(* CoDeSys 2.3.9.41 project: example.pro *)
(* Libraries: Util.lib 18.5.10 15:14:28, STANDARD.LIB 4.10.05 11:14:46, IECSFC.LIB 13.4.06 15:51:28, SYSLIBTIME.LIB 26.10.21 13:46:42, SYSTASKINFO.LIB 26.10.21 13:46:42, ANALYZATION.LIB 5.10.99 09:05:06, SYSLIBCALLBACK.LIB 26.10.21 13:46:42 *)

(* PLC configuration (modules and I/O channels)
Fast discrete inputs [I_SIMPLE_INPUT] node 0, in %IB0 out %QB0 {ChannellName = Fast discrete inputs; Filtrationtime = 10000}
  AT %IX0.0 [BitInput] Discrete input 1 {ChannellName = Enter name}
  AT %IX0.1 [BitInput] Discrete input 2 {ChannellName = Enter name}
Discrete inputs [ID130] node 1, in %IB1 out %QB1 {ChannellName = Discrete inputs; Filtrationtime_GeneralINP = 16; PinCount = 16}
  discrete_input_first_byte AT %IB1.0 [ByteInput] discrete_input_first_byte {ChannellName = Enter name}
  discrete_input_second_byte AT %IB1.1 [ByteInput] discrete input_second_byte {ChannellName = Enter name}
Fast discrete outputs [OWEN_ID570] node 2, in %IB2 out %QB2 {ChannellName = Fast discrete outputs; SafeValueBool = FALSE; SafeValueBool = FALSE; SafeValueBool = FALSE; SafeValueBool = FALSE}
  hw_run_id1 AT %QX2.0 [BitOutput] Run hot water invertor drive1 {ChannellName = Enter name}
  hw_run_id2 AT %QX2.1 [BitOutput] Run hot water invertor drive2 {ChannellName = Enter name}
  ws_run_id1 AT %QX2.2 [BitOutput] Run water supply invertor drive1 {ChannellName = Enter name}
  ws_run_id2 AT %QX2.3 [BitOutput] Run water supply invertor drive2 {ChannellName = Enter name}
Discrete outputs [ID131] node 3, in %IB3 out %QB3 {ChannellName = Discrete outputs; SafeValueByte = 0; SafeValueByte = 0; SafeValueByteM = 0; PinCount = 24}
  AT %QB3.0 [ByteOutput] 8 discrete outputs {ChannellName = Enter name}
  AT %QB3.1 [ByteOutput] 8 discrete outputs {ChannellName = Enter name}
Special input [ID103] node 4, in %IB4 out %QB4 {ChannellName = Special input}
  AT %IX4.0 [BitInput] Special input {ChannellName = Enter name}
Special output [ID104] node 5, in %IB5 out %QB5 {ChannellName = Special output}
  AT %QX5.0 [BitOutput] Special output {ChannellName = Enter name}
AT %QD6.0 [DWordOutput] Last address {ChannellName = Enter name}
AT %QW6.1 [WordOutput] Last error {ChannellName = Enter name}
RS-485-1 [COM1_USART] node 0, in %IB6.0 out %QB6.0 {ChannellName = RS-485-1; CommunicationSpeed = 115200; Parity = NO PARITY CHECK; BitLength = 8 bits; StopLength = One stop bit; InterfaceType = RS485; FrameOriented = RTU; Timeout = 0; Visibility = No}
AT %QB6.1.0 [ComChannel] Command (0xff - Start) {ChannellName = Enter name}
hw_input_pressure AT %QD6.1.0.0 [FloatOutput] {ChannellName = Enter name}
hw_error_input_pressure AT %QW6.1.1.0 [WordOutput] {ChannellName = Enter name}
hw_output_pressure AT %QD6.1.2.0 [FloatOutput] {ChannellName = Enter name}
hw_error_output_pressure AT %QW6.1.3.0 [WordOutput] {ChannellName = Enter name}
ws_input_pressure AT %QD6.1.4.0 [FloatOutput] {ChannellName = Enter name}
ws_error_input_pressure AT %QW6.1.5.0 [WordOutput] {ChannellName = Enter name}
ws_output_pressure AT %QD6.1.6.0 [FloatOutput] {ChannellName = Enter name}
ws_error_output_pressure AT %QW6.1.7.0 [WordOutput] {ChannellName = Enter name}
ModBus (Master) [MODBUS_MASTER_ID450] node 7, in %IB7 out %QB7 {ChannellName = ModBus (Master); Visibility = No}
  AT %QD7.0 [DWordOutput] Last address {ChannellName = Enter name}
  AT %QW7.1 [WordOutput] Last error {ChannellName = Enter name}
  RS-485-1 [COM1_USART] node 0, in %IB7.0 out %QB7.0 {ChannellName = RS-485-1; CommunicationSpeed = 115200; Parity = NO PARITY CHECK; BitLength = 8 bits; StopLength = One stop bit; InterfaceType = RS485; FrameOriented = RTU; Timeout = 0; Visibility = No}
  Universal Modbus device [ID2000] node 1, in %IB7.1 out %QB7.1 {ChannellName = Universal Modbus device; ModuleIP = 10:0:0:223; ServiceTimeout = 150; TCPport = 502; NetMode = Serial; ModuleSlaveAddress = 32; RequestType = By poll time; PeriodOfService = 100; Visibility = No; RepeatCounter = 0; ByteSequence = Trace_mode}
    AT %QB7.1.0 [ComChannel] Command (0xff - Start) {ChannellName = Enter name}
hw_output_value_id1 AT %QW7.1.0.0 [WordOutput] {ChannellName = Enter name}
hw_output_value_id2 AT %QW7.1.1.0 [WordOutput] {ChannellName = Enter name}
ws_output_value_id1 AT %QW7.1.2.0 [WordOutput] {ChannellName = Enter name}
ws_output_value_id2 AT %QW7.1.3.0 [WordOutput] {ChannellName = Enter name}
AT %QW7.1.4.0 [WordOutput] {ChannellName = Enter name}
AT %QW7.1.5.0 [WordOutput] {ChannellName = Enter name}
AT %QW7.1.6.0 [WordOutput] {ChannellName = Enter name}
AT %QW7.1.7.0 [WordOutput] {ChannellName = Enter name}
Modbus [MODBUS_ID302] node 0, in %IB8.0 out %QB8.0 {ChannellName = Modbus}
  RS-232 [COM2_USART] node 0, in %IB8.0.0 out %QB8.0.0 {ChannellName = RS-232; CommunicationSpeed = 115200; Parity = NO PARITY CHECK; BitLength = 8 bits; StopLength = One stop bit; InterfaceType = RS232; FrameOriented = RTU; Timeout = 0; Visibility = No}
8 bits [8Bit] node 1, in %IB8.1 out %QB8.1 {ChannellName = 8 bit}
  AT %QB8.1.0 [ByteOutput] {ChannellName = Enter name}
8 bits [8Bit] node 2, in %IB8.2 out %QB8.2 {ChannellName = 8 bit}
  AT %QB8.2.0 [ByteOutput] {ChannellName = Enter name}
  AT %QB8.3.0 [ByteOutput] {ChannellName = Enter name}
  AT %QB8.4.0 [ByteOutput] {ChannellName = Enter name}
2 byte [Register] node 5, in %IB8.5 out %QB8.5 {ChannellName = 2 byte}
  hw_pivot_single AT %QW8.5.0 [WordOutput] {ChannellName = Enter name}
2 byte [Register] node 6, in %IB8.6 out %QB8.6 {ChannellName = 2 byte}
  hw_pivot_cascade AT %QW8.6.0 [WordOutput] {ChannellName = Enter name}
2 byte [Register] node 7, in %IB8.7 out %QB8.7 {ChannellName = 2 byte}
  hw_cycle_set_hours AT %QW8.7.0 [WordOutput] {ChannellName = Enter name}
2 byte [Register] node 8, in %IB8.8 out %QB8.8 {ChannellName = 2 byte}
  hw_cycle_set_minutes AT %QW8.8.0 [WordOutput] {ChannellName = Enter name}
2 byte [Register] node 9, in %IB8.9 out %QB8.9 {ChannellName = 2 byte}
  hw_cycle_set_seconds AT %QW8.9.0 [WordOutput] {ChannellName = Enter name}
2 byte [Register] node 10, in %IB8.10 out %QB8.10 {ChannellName = 2 byte}
  hw_cascade_delay_on_hours AT %QW8.10.0 [WordOutput] {ChannellName = Enter name}
2 byte [Register] node 11, in %IB8.11 out %QB8.11 {ChannellName = 2 byte}
  hw_cascade_delay_on_minutes AT %QW8.11.0 [WordOutput] {ChannellName = Enter name}
2 byte [Register] node 12, in %IB8.12 out %QB8.12 {ChannellName = 2 byte}
  hw_cascade_delay_on_seconds AT %QW8.12.0 [WordOutput] {ChannellName = Enter name}
2 byte [Register] node 13, in %IB8.13 out %QB8.13 {ChannellName = 2 byte}
  hw_cascade_delay_off_hours AT %QW8.13.0 [WordOutput] {ChannellName = Enter name}
2 byte [Register] node 14, in %IB8.14 out %QB8.14 {ChannellName = 2 byte}
  hw_cascade_delay_off_minutes AT %QW8.14.0 [WordOutput] {ChannellName = Enter name}
2 byte [Register] node 15, in %IB8.15 out %QB8.15 {ChannellName = 2 byte}
  hw_cascade_delay_off_seconds AT %QW8.15.0 [WordOutput] {ChannellName = Enter name}
2 byte [Register] node 16, in %IB8.16 out %QB8.16 {ChannellName = 2 byte}
  ws_pivot_single AT %QW8.16.0 [WordOutput] {ChannellName = Enter name}
2 byte [Register] node 17, in %IB8.17 out %QB8.17 {ChannellName = 2 byte}
  ws_pivot_cascade AT %QW8.17.0 [WordOutput] {ChannellName = Enter name}
2 byte [Register] node 18, in %IB8.18 out %QB8.18 {ChannellName = 2 byte}
  ws_cycle_set_hours AT %QW8.18.0 [WordOutput] {ChannellName = Enter name}
2 byte [Register] node 19, in %IB8.19 out %QB8.19 {ChannellName = 2 byte}
  ws_cycle_set_minutes AT %QW8.19.0 [WordOutput] {ChannellName = Enter name}
2 byte [Register] node 20, in %IB8.20 out %QB8.20 {ChannellName = 2 byte}
  ws_cycle_set_seconds AT %QW8.20.0 [WordOutput] {ChannellName = Enter name}
2 byte [Register] node 21, in %IB8.21 out %QB8.21 {ChannellName = 2 byte}
  ws_cascade_delay_on_hours AT %QW8.21.0 [WordOutput] {ChannellName = Enter name}
2 byte [Register] node 22, in %IB8.22 out %QB8.22 {ChannellName = 2 byte}
  ws_cascade_delay_on_minutes AT %QW8.22.0 [WordOutput] {ChannellName = Enter name}
2 byte [Register] node 23, in %IB8.23 out %QB8.23 {ChannellName = 2 byte}
  ws_cascade_delay_on_seconds AT %QW8.23.0 [WordOutput] {ChannellName = Enter name}
2 byte [Register] node 24, in %IB8.24 out %QB8.24 {ChannellName = 2 byte}
  ws_cascade_delay_off_hours AT %QW8.24.0 [WordOutput] {ChannellName = Enter name}
2 byte [Register] node 25, in %IB8.25 out %QB8.25 {ChannellName = 2 byte}
  ws_cascade_delay_off_minutes AT %QW8.25.0 [WordOutput] {ChannellName = Enter name}
2 byte [Register] node 26, in %IB8.26 out %QB8.26 {ChannellName = 2 byte}
  ws_cascade_delay_off_seconds AT %QW8.26.0 [WordOutput] {ChannellName = Enter name}
Float [Float] node 27, in %IB8.27 out %QB8.27 {ChannellName = float}
  hw_set_point_pressure AT %QD8.27.0 [FloatOutput] {ChannellName = Enter name}
Float [Float] node 28, in %IB8.28 out %QB8.28 {ChannellName = float}
  ws_set_point_pressure AT %QD8.28.0 [FloatOutput] {ChannellName = Enter name}
Float [Float] node 29, in %IB8.29 out %QB8.29 {ChannellName = float}
  hw_min_measure_range_input AT %QD8.29.0 [FloatOutput] {ChannellName = Enter name}
Float [Float] node 30, in %IB8.30 out %QB8.30 {ChannellName = float}
  hw_max_measure_range_input AT %QD8.30.0 [FloatOutput] {ChannellName = Enter name}
Float [Float] node 31, in %IB8.31 out %QB8.31 {ChannellName = float}
  hw_min_measure_range_output AT %QD8.31.0 [FloatOutput] {ChannellName = Enter name}
Float [Float] node 32, in %IB8.32 out %QB8.32 {ChannellName = float}
  hw_max_measure_range_output AT %QD8.32.0 [FloatOutput] {ChannellName = Enter name}
Float [Float] node 33, in %IB8.33 out %QB8.33 {ChannellName = float}
  ws_min_measure_range_input AT %QD8.33.0 [FloatOutput] {ChannellName = Enter name}
Float [Float] node 34, in %IB8.34 out %QB8.34 {ChannellName = float}
  ws_max_measure_range_input AT %QD8.34.0 [FloatOutput] {ChannellName = Enter name}
Float [Float] node 35, in %IB8.35 out %QB8.35 {ChannellName = float}
  ws_min_measure_range_output AT %QD8.35.0 [FloatOutput] {ChannellName = Enter name}
Float [Float] node 36, in %IB8.36 out %QB8.36 {ChannellName = float}
  ws_max_measure_range_output AT %QD8.36.0 [FloatOutput] {ChannellName = Enter name}
Float [Float] node 37, in %IB8.37 out %QB8.37 {ChannellName = float}
  hw_input_pressure_bar AT %QD8.37.0 [FloatOutput] {ChannellName = Enter name}
Float [Float] node 38, in %IB8.38 out %QB8.38 {ChannellName = float}
  hw_output_pressure_bar AT %QD8.38.0 [FloatOutput] {ChannellName = Enter name}
Float [Float] node 39, in %IB8.39 out %QB8.39 {ChannellName = float}
  ws_input_pressure_bar AT %QD8.39.0 [FloatOutput] {ChannellName = Enter name}
Float [Float] node 40, in %IB8.40 out %QB8.40 {ChannellName = float}
  ws_output_pressure_bar AT %QD8.40.0 [FloatOutput] {ChannellName = Enter name}
Float [Float] node 41, in %IB8.41 out %QB8.41 {ChannellName = float}
  hw_frequency_id1 AT %QD8.41.0 [FloatOutput] {ChannellName = Enter name}
Float [Float] node 42, in %IB8.42 out %QB8.42 {ChannellName = float}
  hw_frequency_id2 AT %QD8.42.0 [FloatOutput] {ChannellName = Enter name}
Float [Float] node 43, in %IB8.43 out %QB8.43 {ChannellName = float}
  ws_frequency_id1 AT %QD8.43.0 [FloatOutput] {ChannellName = Enter name}
Float [Float] node 44, in %IB8.44 out %QB8.44 {ChannellName = float}
  ws_frequency_id2 AT %QD8.44.0 [FloatOutput] {ChannellName = Enter name}
2 byte [Register] node 45, in %IB8.45 out %QB8.45 {ChannellName = 2 byte}
  hw_alarm_error_code AT %QW8.45.0 [WordOutput] {ChannellName = Enter name}
2 byte [Register] node 46, in %IB8.46 out %QB8.46 {ChannellName = 2 byte}
  ws_alarm_error_code AT %QW8.46.0 [WordOutput] {ChannellName = Enter name}
Float [Float] node 47, in %IB8.47 out %QB8.47 {ChannellName = float}
  hw_manual_set_frequency_id1 AT %QD8.47.0 [FloatOutput] {ChannellName = Enter name}
Float [Float] node 48, in %IB8.48 out %QB8.48 {ChannellName = float}
  hw_manual_set_frequency_id2 AT %QD8.48.0 [FloatOutput] {ChannellName = Enter name}
Float [Float] node 49, in %IB8.49 out %QB8.49 {ChannellName = float}
  ws_manual_set_frequency_id1 AT %QD8.49.0 [FloatOutput] {ChannellName = Enter name}
Float [Float] node 50, in %IB8.50 out %QB8.50 {ChannellName = float}
  ws_manual_set_frequency_id2 AT %QD8.50.0 [FloatOutput] {ChannellName = Enter name}
2 byte [Register] node 51, in %IB8.51 out %QB8.51 {ChannellName = 2 byte}
  AT %QW8.51.0 [WordOutput] {ChannellName = Enter name}
2 byte [Register] node 52, in %IB8.52 out %QB8.52 {ChannellName = 2 byte}
  AT %QW8.52.0 [WordOutput] {ChannellName = Enter name}
2 byte [Register] node 53, in %IB8.53 out %QB8.53 {ChannellName = 2 byte}
  AT %QW8.53.0 [WordOutput] {ChannellName = Enter name}
2 byte [Register] node 54, in %IB8.54 out %QB8.54 {ChannellName = 2 byte}
  AT %QW8.54.0 [WordOutput] {ChannellName = Enter name}
2 byte [Register] node 55, in %IB8.55 out %QB8.55 {ChannellName = 2 byte}
  AT %QW8.55.0 [WordOutput] {ChannellName = Enter name}
2 byte [Register] node 56, in %IB8.56 out %QB8.56 {ChannellName = 2 byte}
  AT %QW8.56.0 [WordOutput] {ChannellName = Enter name}
2 byte [Register] node 57, in %IB8.57 out %QB8.57 {ChannellName = 2 byte}
  AT %QW8.57.0 [WordOutput] {ChannellName = Enter name}
2 byte [Register] node 58, in %IB8.58 out %QB8.58 {ChannellName = 2 byte}
  AT %QW8.58.0 [WordOutput] {ChannellName = Enter name}
2 byte [Register] node 59, in %IB8.59 out %QB8.59 {ChannellName = 2 byte}
  AT %QW8.59.0 [WordOutput] {ChannellName = Enter name}
2 byte [Register] node 60, in %IB8.60 out %QB8.60 {ChannellName = 2 byte}
  AT %QW8.60.0 [WordOutput] {ChannellName = Enter name}
2 byte [Register] node 61, in %IB8.61 out %QB8.61 {ChannellName = 2 byte}
  AT %QW8.61.0 [WordOutput] {ChannellName = Enter name}
2 byte [Register] node 62, in %IB8.62 out %QB8.62 {ChannellName = 2 byte}
  AT %QW8.62.0 [WordOutput] {ChannellName = Enter name}
2 byte [Register] node 63, in %IB8.63 out %QB8.63 {ChannellName = 2 byte}
  AT %QW8.63.0 [WordOutput] {ChannellName = Enter name}
2 byte [Register] node 64, in %IB8.64 out %QB8.64 {ChannellName = 2 byte}
  AT %QW8.64.0 [WordOutput] {ChannellName = Enter name}
2 byte [Register] node 65, in %IB8.65 out %QB8.65 {ChannellName = 2 byte}
  AT %QW8.65.0 [WordOutput] {ChannellName = Enter name}
2 byte [Register] node 66, in %IB8.66 out %QB8.66 {ChannellName = 2 byte}
  AT %QW8.66.0 [WordOutput] {ChannellName = Enter name}
2 byte [Register] node 67, in %IB8.67 out %QB8.67 {ChannellName = 2 byte}
  AT %QW8.67.0 [WordOutput] {ChannellName = Enter name}
2 byte [Register] node 68, in %IB8.68 out %QB8.68 {ChannellName = 2 byte}
  AT %QW8.68.0 [WordOutput] {ChannellName = Enter name}
2 byte [Register] node 69, in %IB8.69 out %QB8.69 {ChannellName = 2 byte}
  AT %QW8.69.0 [WordOutput] {ChannellName = Enter name}
2 byte [Register] node 70, in %IB8.70 out %QB8.70 {ChannellName = 2 byte}
  AT %QW8.70.0 [WordOutput] {ChannellName = Enter name}
2 byte [Register] node 71, in %IB8.71 out %QB8.71 {ChannellName = 2 byte}
  AT %QW8.71.0 [WordOutput] {ChannellName = Enter name}
2 byte [Register] node 72, in %IB8.72 out %QB8.72 {ChannellName = 2 byte}
  AT %QW8.72.0 [WordOutput] {ChannellName = Enter name}
2 byte [Register] node 73, in %IB8.73 out %QB8.73 {ChannellName = 2 byte}
  AT %QW8.73.0 [WordOutput] {ChannellName = Enter name}
2 byte [Register] node 74, in %IB8.74 out %QB8.74 {ChannellName = 2 byte}
  AT %QW8.74.0 [WordOutput] {ChannellName = Enter name}
2 byte [Register] node 75, in %IB8.75 out %QB8.75 {ChannellName = 2 byte}
  AT %QW8.75.0 [WordOutput] {ChannellName = Enter name}
2 byte [Register] node 76, in %IB8.76 out %QB8.76 {ChannellName = 2 byte}
  AT %QW8.76.0 [WordOutput] {ChannellName = Enter name}
2 byte [Register] node 77, in %IB8.77 out %QB8.77 {ChannellName = 2 byte}
  AT %QW8.77.0 [WordOutput] {ChannellName = Enter name}
2 byte [Register] node 78, in %IB8.78 out %QB8.78 {ChannellName = 2 byte}
  AT %QW8.78.0 [WordOutput] {ChannellName = Enter name}
2 byte [Register] node 79, in %IB8.79 out %QB8.79 {ChannellName = 2 byte}
  AT %QW8.79.0 [WordOutput] {ChannellName = Enter name}
2 byte [Register] node 80, in %IB8.80 out %QB8.80 {ChannellName = 2 byte}
  AT %QW8.80.0 [WordOutput] {ChannellName = Enter name}
2 byte [Register] node 81, in %IB8.81 out %QB8.81 {ChannellName = 2 byte}
  AT %QW8.81.0 [WordOutput] {ChannellName = Enter name}
2 byte [Register] node 82, in %IB8.82 out %QB8.82 {ChannellName = 2 byte}
  AT %QW8.82.0 [WordOutput] {ChannellName = Enter name}
2 byte [Register] node 83, in %IB8.83 out %QB8.83 {ChannellName = 2 byte}
  AT %QW8.83.0 [WordOutput] {ChannellName = Enter name}
2 byte [Register] node 84, in %IB8.84 out %QB8.84 {ChannellName = 2 byte}
  AT %QW8.84.0 [WordOutput] {ChannellName = Enter name}
2 byte [Register] node 85, in %IB8.85 out %QB8.85 {ChannellName = 2 byte}
  AT %QW8.85.0 [WordOutput] {ChannellName = Enter name}
2 byte [Register] node 86, in %IB8.86 out %QB8.86 {ChannellName = 2 byte}
  AT %QW8.86.0 [WordOutput] {ChannellName = Enter name}
2 byte [Register] node 87, in %IB8.87 out %QB8.87 {ChannellName = 2 byte}
  AT %QW8.87.0 [WordOutput] {ChannellName = Enter name}
2 byte [Register] node 88, in %IB8.88 out %QB8.88 {ChannellName = 2 byte}
  AT %QW8.88.0 [WordOutput] {ChannellName = Enter name}
2 byte [Register] node 89, in %IB8.89 out %QB8.89 {ChannellName = 2 byte}
  AT %QW8.89.0 [WordOutput] {ChannellName = Enter name}
2 byte [Register] node 90, in %IB8.90 out %QB8.90 {ChannellName = 2 byte}
  AT %QW8.90.0 [WordOutput] {ChannellName = Enter name}
2 byte [Register] node 91, in %IB8.91 out %QB8.91 {ChannellName = 2 byte}
  AT %QW8.91.0 [WordOutput] {ChannellName = Enter name}
2 byte [Register] node 92, in %IB8.92 out %QB8.92 {ChannellName = 2 byte}
  AT %QW8.92.0 [WordOutput] {ChannellName = Enter name}
2 byte [Register] node 93, in %IB8.93 out %QB8.93 {ChannellName = 2 byte}
  AT %QW8.93.0 [WordOutput] {ChannellName = Enter name}
2 byte [Register] node 94, in %IB8.94 out %QB8.94 {ChannellName = 2 byte}
  AT %QW8.94.0 [WordOutput] {ChannellName = Enter name}
2 byte [Register] node 95, in %IB8.95 out %QB8.95 {ChannellName = 2 byte}
  AT %QW8.95.0 [WordOutput] {ChannellName = Enter name}
2 byte [Register] node 96, in %IB8.96 out %QB8.96 {ChannellName = 2 byte}
  AT %QW8.96.0 [WordOutput] {ChannellName = Enter name}
2 byte [Register] node 97, in %IB8.97 out %QB8.97 {ChannellName = 2 byte}
  AT %QW8.97.0 [WordOutput] {ChannellName = Enter name}
2 byte [Register] node 98, in %IB8.98 out %QB8.98 {ChannellName = 2 byte}
  AT %QW8.98.0 [WordOutput] {ChannellName = Enter name}
2 byte [Register] node 99, in %IB8.99 out %QB8.99 {ChannellName = 2 byte}
  AT %QW8.99.0 [WordOutput] {ChannellName = Enter name}
2 byte [Register] node 100, in %IB8.100 out %QB8.100 {ChannellName = 2 byte}
  AT %QW8.100.0 [WordOutput] {ChannellName = Enter name}
2 byte [Register] node 101, in %IB8.101 out %QB8.101 {ChannellName = 2 byte}
  AT %QW8.101.0 [WordOutput] {ChannellName = Enter name}
2 byte [Register] node 102, in %IB8.102 out %QB8.102 {ChannellName = 2 byte}
  AT %QW8.102.0 [WordOutput] {ChannellName = Enter name}
2 byte [Register] node 103, in %IB8.103 out %QB8.103 {ChannellName = 2 byte}
  AT %QW8.103.0 [WordOutput] {ChannellName = Enter name}
2 byte [Register] node 104, in %IB8.104 out %QB8.104 {ChannellName = 2 byte}
  AT %QW8.104.0 [WordOutput] {ChannellName = Enter name}
2 byte [Register] node 105, in %IB8.105 out %QB8.105 {ChannellName = 2 byte}
  AT %QW8.105.0 [WordOutput] {ChannellName = Enter name}
2 byte [Register] node 106, in %IB8.106 out %QB8.106 {ChannellName = 2 byte}
  AT %QW8.106.0 [WordOutput] {ChannellName = Enter name}
2 byte [Register] node 107, in %IB8.107 out %QB8.107 {ChannellName = 2 byte}
  AT %QW8.107.0 [WordOutput] {ChannellName = Enter name}
2 byte [Register] node 108, in %IB8.108 out %QB8.108 {ChannellName = 2 byte}
  AT %QW8.108.0 [WordOutput] {ChannellName = Enter name}
2 byte [Register] node 109, in %IB8.109 out %QB8.109 {ChannellName = 2 byte}
  AT %QW8.109.0 [WordOutput] {ChannellName = Enter name}
2 byte [Register] node 110, in %IB8.110 out %QB8.110 {ChannellName = 2 byte}
  AT %QW8.110.0 [WordOutput] {ChannellName = Enter name}
2 byte [Register] node 111, in %IB8.111 out %QB8.111 {ChannellName = 2 byte}
  AT %QW8.111.0 [WordOutput] {ChannellName = Enter name}
2 byte [Register] node 112, in %IB8.112 out %QB8.112 {ChannellName = 2 byte}
  AT %QW8.112.0 [WordOutput] {ChannellName = Enter name}
2 byte [Register] node 113, in %IB8.113 out %QB8.113 {ChannellName = 2 byte}
  AT %QW8.113.0 [WordOutput] {ChannellName = Enter name}
2 byte [Register] node 114, in %IB8.114 out %QB8.114 {ChannellName = 2 byte}
  AT %QW8.114.0 [WordOutput] {ChannellName = Enter name}
2 byte [Register] node 115, in %IB8.115 out %QB8.115 {ChannellName = 2 byte}
  AT %QW8.115.0 [WordOutput] {ChannellName = Enter name}
2 byte [Register] node 116, in %IB8.116 out %QB8.116 {ChannellName = 2 byte}
  AT %QW8.116.0 [WordOutput] {ChannellName = Enter name}
2 byte [Register] node 117, in %IB8.117 out %QB8.117 {ChannellName = 2 byte}
  AT %QW8.117.0 [WordOutput] {ChannellName = Enter name}
2 byte [Register] node 118, in %IB8.118 out %QB8.118 {ChannellName = 2 byte}
  AT %QW8.118.0 [WordOutput] {ChannellName = Enter name}
2 byte [Register] node 119, in %IB8.119 out %QB8.119 {ChannellName = 2 byte}
  AT %QW8.119.0 [WordOutput] {ChannellName = Enter name}
2 byte [Register] node 120, in %IB8.120 out %QB8.120 {ChannellName = 2 byte}
  AT %QW8.120.0 [WordOutput] {ChannellName = Enter name}
2 byte [Register] node 121, in %IB8.121 out %QB8.121 {ChannellName = 2 byte}
  AT %QW8.121.0 [WordOutput] {ChannellName = Enter name}
2 byte [Register] node 122, in %IB8.122 out %QB8.122 {ChannellName = 2 byte}
  AT %QW8.122.0 [WordOutput] {ChannellName = Enter name}
2 byte [Register] node 123, in %IB8.123 out %QB8.123 {ChannellName = 2 byte}
  AT %QW8.123.0 [WordOutput] {ChannellName = Enter name}
2 byte [Register] node 124, in %IB8.124 out %QB8.124 {ChannellName = 2 byte}
  AT %QW8.124.0 [WordOutput] {ChannellName = Enter name}
2 byte [Register] node 125, in %IB8.125 out %QB8.125 {ChannellName = 2 byte}
  AT %QW8.125.0 [WordOutput] {ChannellName = Enter name}
2 byte [Register] node 126, in %IB8.126 out %QB8.126 {ChannellName = 2 byte}
  AT %QW8.126.0 [WordOutput] {ChannellName = Enter name}
2 byte [Register] node 127, in %IB8.127 out %QB8.127 {ChannellName = 2 byte}
  AT %QW8.127.0 [WordOutput] {ChannellName = Enter name}
2 byte [Register] node 128, in %IB8.128 out %QB8.128 {ChannellName = 2 byte}
  AT %QW8.128.0 [WordOutput] {ChannellName = Enter name}
2 byte [Register] node 129, in %IB8.129 out %QB8.129 {ChannellName = 2 byte}
  AT %QW8.129.0 [WordOutput] {ChannellName = Enter name}
2 byte [Register] node 130, in %IB8.130 out %QB8.130 {ChannellName = 2 byte}
  AT %QW8.130.0 [WordOutput] {ChannellName = Enter name}
2 byte [Register] node 131, in %IB8.131 out %QB8.131 {ChannellName = 2 byte}
  AT %QW8.131.0 [WordOutput] {ChannellName = Enter name}
*)

(* Data type in InvertorDrive *)
TYPE classAlarmInvertorDrive :

STRUCT
	external_alarm:STRING(79);
	fault_invertor_drive:STRING(79);
END_STRUCT

END_TYPE

(* Data type in MB110_8U *)
TYPE classAnalogOutputChannel :

STRUCT
	current_value: REAL;
END_STRUCT

END_TYPE

(* Data type in MB110_8U *)
TYPE classAnalogOutputModule :

STRUCT
	channel1:classAnalogOutputChannel;
	channel2:classAnalogOutputChannel;
	channel3:classAnalogOutputChannel;
	channel4:classAnalogOutputChannel;
	channel5:classAnalogOutputChannel;
	channel6:classAnalogOutputChannel;
	channel7:classAnalogOutputChannel;
	channel8:classAnalogOutputChannel;
END_STRUCT

END_TYPE

(* Data type in PLC110/DiscreteInputs *)
TYPE classDiscreteInputByte :

STRUCT
	Bit1:BOOL;
	Bit2:BOOL;
	Bit3:BOOL;
	Bit4:BOOL;
	Bit5:BOOL;
	Bit6:BOOL;
	Bit7:BOOL;
	Bit8:BOOL;
END_STRUCT

END_TYPE

(* Data type in PLC110/DiscreteInputs *)
TYPE classDiscreteInputs :

STRUCT
	first_byte:classDiscreteInputByte;
	second_byte:classDiscreteInputByte;
END_STRUCT

END_TYPE

(* Data type in PLC110/DiscreteOutputs *)
TYPE classDiscreteOutputByte :

STRUCT
	Bit1:BOOL;
	Bit2:BOOL;
	Bit3:BOOL;
	Bit4:BOOL;
	Bit5:BOOL;
	Bit6:BOOL;
	Bit7:BOOL;
	Bit8:BOOL;
END_STRUCT

END_TYPE

(* Data type in PLC110/DiscreteOutputs *)
TYPE classDiscreteOutputs :

STRUCT
	first_byte:classDiscreteOutputByte;
	second_byte:classDiscreteOutputByte;
END_STRUCT

END_TYPE

(* Data type in PLC110/DiscreteInputs *)
TYPE classFastDiscreteInputs :

STRUCT
	Bit1:BOOL;
	Bit2:BOOL;
END_STRUCT

END_TYPE

(* Data type in PLC110/DiscreteOutputs *)
TYPE classFastDiscreteOutputs :

STRUCT
	Bit1:BOOL;
	Bit2:BOOL;
	Bit3:BOOL;
	Bit4:BOOL;
END_STRUCT

END_TYPE

(* Data type in MB110_8A *)
TYPE classInfoAnalogInputChannel :

STRUCT
	current_value:REAL;
	error_message:STRING(79);
END_STRUCT

END_TYPE

(* Data type in MB110_8A *)
TYPE classInfoAnalogInputModule :

STRUCT
	channel1:classInfoAnalogInputChannel;
	channel2:classInfoAnalogInputChannel;
	channel3:classInfoAnalogInputChannel;
	channel4:classInfoAnalogInputChannel;
	channel5:classInfoAnalogInputChannel;
	channel6:classInfoAnalogInputChannel;
	channel7:classInfoAnalogInputChannel;
	channel8:classInfoAnalogInputChannel;
END_STRUCT

END_TYPE

(* Data type in CascadeMode *)
TYPE classInfoCascade :

STRUCT
	pivot:INT;
	error_message:STRING(79);
	error_code: WORD;
	cascade_pump1:classInfoCascadePump;
	cascade_pump2:classInfoCascadePump;
	cascade_pump3:classInfoCascadePump;
	cascade_pump4:classInfoCascadePump;
	cascade_pump5:classInfoCascadePump;
	cascade_pump6:classInfoCascadePump;
	cascade_pump7:classInfoCascadePump;
	cascade_pump8:classInfoCascadePump;
END_STRUCT

END_TYPE

(* Data type in CascadeMode *)
TYPE classInfoCascadePump :

STRUCT
	cascade_pump:BOOL := FALSE;  (*ï¿½ï¿½ï¿½ï¿½ï¿½ï¿½ ï¿½ï¿½ï¿½ï¿½ï¿½ï¿½ ï¿½ï¿½ï¿½ï¿½ï¿½ï¿½*)
	manual:INT := 40;  (*Hz*)
END_STRUCT

END_TYPE

(* Data type in CycleMode *)
TYPE classInfoCycle :

STRUCT
	run_timer: BOOL; (* status work *)
	working_time: TIME; (* pump working time  *)
	pump_number: INT;  (* number working pump *)
	error_code:  WORD;
END_STRUCT

END_TYPE

(* Data type in InvertorDrive *)
TYPE classInfoInvertorDrive :

STRUCT
	active:BOOL;
	status_run:STRING(79);
	set_pid:classSetPid;
	alarm:classAlarmInvertorDrive;
	frequency:REAL;  (* Hz *)
	aout_frequency:REAL;  (* mA *)
	run:BOOL;
	reset_fault:BOOL;
END_STRUCT

END_TYPE

(* Data type in SingleMode *)
TYPE classInfoSingle :
(* class for information single mode. *)

STRUCT
    pivot_pump : INT;
    start_pump : BOOL;
    message: STRING(79);
    error_code: WORD;
END_STRUCT

END_TYPE

(* Data type in InvertorDrive *)
TYPE classInvertorDrive :

STRUCT
	discrete_inputs:classInvertorDriveDiscreteInputs;
	discrete_outputs:classInvertorDriveDiscreteOutputs;
	analog_input:classInvertorDriveAnalogInputs;
	analog_output:classInvertorDriveAnalogOutputs;
	set:classSetInvertorDrive;
	min_frequency:INT;
	max_frequency:INT;
	set_frequency:REAL;
	real_frequency:REAL;(* ï¿½ï¿½ï¿½ï¿½ï¿½ï¿½ï¿½ï¿½ ï¿½ ï¿½ï¿½ï¿½ï¿½ï¿½ï¿½ï¿½ï¿½ï¿½ï¿½ï¿½ ï¿½ï¿½ï¿½ï¿½ï¿½ï¿½ ï¿½ï¿½ï¿½ï¿½ï¿½ï¿½ï¿½ï¿½ï¿½ï¿½ *)
END_STRUCT

END_TYPE

(* Data type in InvertorDrive *)
TYPE classInvertorDriveAnalogInputs :

STRUCT
	set_frequency:REAL;
END_STRUCT

END_TYPE

(* Data type in InvertorDrive *)
TYPE classInvertorDriveAnalogOutputs :

STRUCT
	out_frequency:REAL;
END_STRUCT

END_TYPE

(* Data type in InvertorDrive *)
TYPE classInvertorDriveDiscreteInputs :

STRUCT
	start:BOOL;
	reset_fault:BOOL;
(* external alarm *)
	low_pressure_in:BOOL;
	high_pressure_out:BOOL;
END_STRUCT

END_TYPE

(* Data type in InvertorDrive *)
TYPE classInvertorDriveDiscreteOutputs :

STRUCT
	status_run:BOOL;
	status_alarm:BOOL;
END_STRUCT

END_TYPE

(* Data type in value_scale *)
TYPE classParamsValueScaling :

STRUCT
	in_min: REAL := 0;
	in_max: REAL := 100;
	out_min: REAL := 0;
	out_max: REAL := 100;

END_STRUCT

END_TYPE

(* Data type in PLC110 *)
TYPE classPLC110_32 :

STRUCT
	fast_discrete_inputs:classFastDiscreteInputs;
	discrete_inputs:classDiscreteInputs;
	special_input:classSpecialInput;
	fast_discrete_outputs:classFastDiscreteOutputs;
	discrete_output:classDiscreteOutputs;
	special_output:classSpecialOutput;
END_STRUCT

END_TYPE

(* Data type in PLC110 *)
TYPE classPLC32m2StatusInputs :

STRUCT
	fast_inputs:classFastDiscreteInputs;
	discrete_inputs:classDiscreteInputs;
	special_input:classSpecialInput;
END_STRUCT

END_TYPE

(* Data type in PLC110 *)
TYPE classPLC32m2StatusOutputs :

STRUCT
	fast_outputs:classFastDiscreteOutputs;
	discrete_outputs:classDiscreteOutputs;
	special_output:classSpecialOutput;
END_STRUCT

END_TYPE

(* Data type in MB110_8A *)
TYPE classSetAnalogInputChannel :

STRUCT
	(* ï¿½ï¿½ï¿½ï¿½ï¿½ï¿½ï¿½ï¿½ï¿½ï¿½ï¿½ï¿½ï¿½ï¿½ï¿½ï¿½ ï¿½ï¿½ï¿½ï¿½ï¿½ï¿½ï¿½ï¿½ï¿½ ï¿½ï¿½ï¿½ï¿½ï¿½ï¿½ ï¿½ï¿½ï¿½ï¿½ï¿½ï¿½. ï¿½ï¿½. ï¿½ï¿½ï¿½ï¿½ï¿½ï¿½ï¿½ï¿½ï¿½ï¿½ ï¿½ï¿½ï¿½ï¿½ï¿½ï¿½ï¿½: ï¿½ï¿½ï¿½ï¿½ï¿½ï¿½ï¿½ï¿½ï¿½ï¿½. ï¿½ï¿½ï¿½ï¿½ï¿½ï¿½ï¿½ ï¿½.2 *)
	(* ï¿½ï¿½ï¿½ï¿½ï¿½ï¿½ï¿½ ï¿½ï¿½ï¿½ ï¿½ ï¿½ï¿½ï¿½ï¿½ï¿½ï¿½ï¿½ï¿½ ï¿½ï¿½ ï¿½ï¿½ï¿½ï¿½ï¿½ï¿½ï¿½ï¿½ï¿½: ï¿½ï¿½ï¿½ ï¿½ï¿½ï¿½ï¿½ï¿½ï¿½ï¿½ 4-20mA  *)
	ain_l: REAL := 0;  (* ï¿½ï¿½ï¿½ï¿½ï¿½ï¿½ï¿½ï¿½ Ain.L *)
	ain_h: REAL := 1000;  (* ï¿½ï¿½ï¿½ï¿½ï¿½ï¿½ï¿½ï¿½ Ain.H *)
	analog_min_value: REAL := 4;  (* ï¿½ï¿½ï¿½ï¿½ï¿½ï¿½ï¿½ï¿½ ï¿½ï¿½ï¿½ï¿½ï¿½ï¿½ ï¿½ï¿½ï¿½ï¿½ï¿½ï¿½ï¿½ ï¿½ï¿½ï¿½ï¿½ï¿½ï¿½ï¿½ ï¿½ï¿½ï¿½ï¿½ï¿½ï¿½ï¿½ï¿½ *)
	analog_max_value: REAL := 20;  (* ï¿½ï¿½ï¿½ï¿½ï¿½ï¿½ï¿½ï¿½ ï¿½ï¿½ï¿½ï¿½ï¿½ï¿½ï¿½ ï¿½ï¿½ï¿½ï¿½ï¿½ï¿½ï¿½ ï¿½ï¿½ï¿½ï¿½ï¿½ï¿½ï¿½ ï¿½ï¿½ï¿½ï¿½ï¿½ï¿½ï¿½ï¿½ *)
END_STRUCT

END_TYPE

(* Data type in MB110_8A *)
TYPE classSetAnalogInputsModule :

STRUCT
	ch1_set:classSetAnalogInputChannel;
	ch2_set:classSetAnalogInputChannel;
	ch3_set:classSetAnalogInputChannel;
	ch4_set:classSetAnalogInputChannel;
	ch5_set:classSetAnalogInputChannel;
	ch6_set:classSetAnalogInputChannel;
	ch7_set:classSetAnalogInputChannel;
	ch8_set:classSetAnalogInputChannel;
END_STRUCT

END_TYPE

(* Data type in InvertorDrive/set_auto_invertor_drive *)
TYPE classSetAutoInvertorDrive :

STRUCT
	auto:BOOL := FALSE;
	direct_logic:BOOL := TRUE;  (* ï¿½ï¿½ï¿½ï¿½ ï¿½ï¿½ï¿½ï¿½ï¿½ï¿½ï¿½/ï¿½ï¿½ï¿½ï¿½ï¿½ï¿½ï¿½ï¿½ï¿½ ï¿½ï¿½ï¿½ï¿½ï¿½ï¿½ï¿½ï¿½ï¿½ï¿½; ï¿½ï¿½ï¿½ ï¿½ï¿½ï¿½ï¿½ï¿½ï¿½ï¿½ï¿½ ï¿½ï¿½ï¿½ï¿½ï¿½ï¿½ï¿½ï¿½ï¿½ï¿½ ï¿½ï¿½ï¿½ï¿½ ï¿½ï¿½ï¿½ï¿½ï¿½ï¿½ï¿½ï¿½ ï¿½ï¿½ï¿½ï¿½ï¿½ï¿½ï¿½ï¿½ï¿½ï¿½ï¿½ï¿½ï¿½ï¿½ ï¿½ï¿½ï¿½ï¿½ï¿½ï¿½ï¿½ï¿½ ï¿½ï¿½ï¿½ï¿½ ï¿½ï¿½ï¿½ï¿½ï¿½ï¿½ï¿½, ï¿½ï¿½ï¿½ï¿½ï¿½ï¿½ï¿½ï¿½ ï¿½ï¿½ï¿½ï¿½ï¿½ï¿½ï¿½ ï¿½ï¿½ï¿½ï¿½ï¿½ï¿½ï¿½ï¿½ï¿½ï¿½ï¿½, ï¿½ ï¿½ï¿½ï¿½ï¿½ï¿½ï¿½ï¿½ï¿½*)
	set_point:REAL := 0;  (* ï¿½ï¿½ï¿½ï¿½ï¿½ï¿½ï¿½, ï¿½ï¿½ï¿½ï¿½ï¿½ï¿½ï¿½ï¿½ ï¿½ ï¿½ï¿½ï¿½ï¿½ï¿½ï¿½ï¿½ï¿½ ï¿½ï¿½ï¿½ï¿½ï¿½ï¿½ï¿½ï¿½ï¿½ ï¿½ï¿½ï¿½ï¿½ï¿½ï¿½ï¿½ï¿½ï¿½ï¿½ï¿½ï¿½ï¿½ï¿½ ï¿½ï¿½ï¿½ï¿½ï¿½ï¿½ï¿½ï¿½ *)
	value:REAL := 0;  (* ï¿½ï¿½ï¿½ï¿½ï¿½ï¿½ï¿½ ï¿½ï¿½ï¿½ï¿½ï¿½ï¿½ï¿½ï¿½ ï¿½ï¿½ï¿½ï¿½ï¿½ï¿½ï¿½ï¿½ï¿½ï¿½ï¿½ï¿½ï¿½ï¿½ ï¿½ï¿½ï¿½ï¿½ï¿½ï¿½ï¿½ï¿½, ï¿½ï¿½ï¿½ï¿½ï¿½ï¿½ï¿½ï¿½ï¿½ï¿½ ï¿½ ï¿½ï¿½ï¿½ï¿½ï¿½ï¿½ï¿½ *)
	P:REAL := 2;  (* ï¿½ï¿½ï¿½ï¿½ï¿½ï¿½ï¿½ï¿½ï¿½ï¿½ï¿½ï¿½ï¿½ï¿½ï¿½ï¿½ ï¿½ï¿½ï¿½ï¿½ï¿½ï¿½ï¿½ï¿½ï¿½ï¿½ï¿½ ï¿½ï¿½ï¿½ï¿½ï¿½ï¿½ï¿½ï¿½ï¿½ï¿½, ï¿½ï¿½ï¿½ ï¿½ï¿½ï¿½ï¿½ï¿½ï¿½ï¿½ï¿½ï¿½ï¿½ ï¿½ï¿½ï¿½ï¿½ï¿½ ï¿½ï¿½ï¿½ï¿½ï¿½ï¿½ï¿½ï¿½ï¿½ï¿½ ï¿½ï¿½ï¿½ï¿½ï¿½ï¿½ï¿½ï¿½ï¿½ï¿½ ï¿½ï¿½ï¿½ï¿½ï¿½ï¿½ï¿½*)
	I:INT := 10;  (* ï¿½ï¿½ï¿½ï¿½ï¿½ï¿½ï¿½ï¿½ï¿½ï¿½ï¿½ï¿½ ï¿½ï¿½ï¿½ï¿½ï¿½ï¿½ï¿½ï¿½ï¿½ï¿½ï¿½ ï¿½ï¿½ï¿½ï¿½ï¿½ï¿½ï¿½ï¿½ï¿½ï¿½, ï¿½ï¿½ï¿½ï¿½ï¿½ ï¿½ ï¿½ï¿½ï¿½ï¿½ï¿½ï¿½ï¿½ï¿½ *)
	D:INT := 0;  (* ï¿½ï¿½ï¿½ï¿½ï¿½ï¿½ï¿½ï¿½ï¿½ï¿½ï¿½ï¿½ï¿½ï¿½ï¿½ï¿½ ï¿½ï¿½ï¿½ï¿½ï¿½ï¿½ï¿½ï¿½ï¿½ï¿½ï¿½ ï¿½ï¿½ï¿½ï¿½ï¿½ï¿½ï¿½ï¿½ï¿½ï¿½, ï¿½ï¿½ï¿½ï¿½ï¿½ ï¿½ ï¿½ï¿½ï¿½ï¿½ï¿½ï¿½ï¿½ï¿½ *)
END_STRUCT

END_TYPE

(* Data type in InvertorDrive *)
TYPE classSetInvertorDrive :

STRUCT
	set_auto:classSetAutoInvertorDrive;
	set_frequency:classSetLimitFrequency;
END_STRUCT

END_TYPE

(* Data type in InvertorDrive/set_limit_frequency *)
TYPE classSetLimitFrequency :

STRUCT
	manual:REAL;  (* Hz *)
	min_range:REAL;  (* Hz *)
	max_range:REAL;  (* Hz *)
END_STRUCT

END_TYPE

(* Data type in PID_regulator *)
TYPE classSetPid :

STRUCT
	actual:REAL;
	set_point:REAL;
	P:REAL;  (* ï¿½ï¿½ï¿½ï¿½ï¿½ï¿½ï¿½ï¿½ï¿½ï¿½ï¿½ï¿½ï¿½ï¿½ï¿½ï¿½ ï¿½ï¿½ï¿½ï¿½ï¿½ï¿½ï¿½ï¿½ï¿½ï¿½ï¿½ ï¿½ï¿½ï¿½ï¿½ï¿½ï¿½ï¿½ï¿½ï¿½ï¿½, ï¿½ï¿½ï¿½ ï¿½ï¿½ï¿½ï¿½ï¿½ï¿½ï¿½ï¿½ï¿½ï¿½ ï¿½ï¿½ï¿½ï¿½ï¿½ ï¿½ï¿½ï¿½ï¿½ï¿½ï¿½ï¿½ï¿½ï¿½ï¿½ ï¿½ï¿½ï¿½ï¿½ï¿½ï¿½ï¿½ï¿½ï¿½ï¿½ ï¿½ï¿½ï¿½ï¿½ï¿½ï¿½ï¿½*)
	I:INT;  (* ï¿½ï¿½ï¿½ï¿½ï¿½ï¿½ï¿½ï¿½ï¿½ï¿½ï¿½ï¿½ ï¿½ï¿½ï¿½ï¿½ï¿½ï¿½ï¿½ï¿½ï¿½ï¿½ï¿½ ï¿½ï¿½ï¿½ï¿½ï¿½ï¿½ï¿½ï¿½ï¿½ï¿½, ï¿½ï¿½ï¿½ï¿½ï¿½ ï¿½ ï¿½ï¿½ï¿½ï¿½ï¿½ï¿½ï¿½ï¿½ *)
	D:INT;  (* ï¿½ï¿½ï¿½ï¿½ï¿½ï¿½ï¿½ï¿½ï¿½ï¿½ï¿½ï¿½ï¿½ï¿½ï¿½ï¿½ ï¿½ï¿½ï¿½ï¿½ï¿½ï¿½ï¿½ï¿½ï¿½ï¿½ï¿½ ï¿½ï¿½ï¿½ï¿½ï¿½ï¿½ï¿½ï¿½ï¿½ï¿½, ï¿½ï¿½ï¿½ï¿½ï¿½ ï¿½ ï¿½ï¿½ï¿½ï¿½ï¿½ï¿½ï¿½ï¿½ *)
	Y_manual:REAL := 0;
	Y_offset:REAL;
	Y_min:REAL;
	Y_max:REAL;
	manual:BOOL;
	reset:BOOL;
END_STRUCT

END_TYPE

(* Data type in PressureSensor_4_20ma *)
TYPE classSetPressureSensor4_20 :

STRUCT
	min_measure_range:REAL:=0;
	max_measure_range:REAL:=16;
	min_current_range:REAL:=4;
	max_current_range:REAL:=20;
END_STRUCT

END_TYPE

(* Data type in PLC110/DiscreteInputs *)
TYPE classSpecialInput :

STRUCT
	Bit1:BOOL;
END_STRUCT

END_TYPE

(* Data type in PLC110/DiscreteOutputs *)
TYPE classSpecialOutput :

STRUCT
	Bit1:BOOL;
END_STRUCT

END_TYPE

(* POU PLC_PRG, CFC *)
PROGRAM PLC_PRG
VAR
	PLC: PLC110_32m2;
	analog_inputs_module: MB110_8a;
	currents_value_pack: get_info_analog_outputs_module;
	analog_outputs_module: MY110_8u;
	settings_channel_analog_inputs_module: SetChannelsAnalogInputsModule;
	hw_input: CurrentSensorPressure_4_20;
	hw_output: CurrentSensorPressure_4_20;
	ws_input: CurrentSensorPressure_4_20;
	ws_output: CurrentSensorPressure_4_20;
	(*hw_settings_pressure_input: SetCurrentSensorPressure_4_20;
	hw_settings_pressure_output: SetCurrentSensorPressure_4_20;
	ws_settings_pressure_input: SetCurrentSensorPressure_4_20;
	ws_settings_pressure_output: SetCurrentSensorPressure_4_20;*)
	hw_invertor_drive_1: InvertorDrive;
	hw_invertor_drive_2: InvertorDrive;
	ws_invertor_drive_1: InvertorDrive;
	ws_invertor_drive_2: InvertorDrive;
	hw_settings_pid_id_1: params_in_set_PID;
	hw_settings_pid_id_2: params_in_set_PID;
	ws_settings_pid_id_1: params_in_set_PID;
	ws_settings_pid_id_2: params_in_set_PID;
	pid1: PID;
	pid2: PID;
	pid3: PID;
	pid4: PID;
	 hw_frequency_id_1: REAL;
	hw_frequency_id_2: REAL;
	ws_frequency_id_1: REAL;
	ws_frequency_id_2: REAL;
	(* hw_input_pressure_bar: REAL;
	hw_output_pressure_bar: REAL;
	ws_input_pressure_bar: REAL;
	ws_output_pressure_bar: REAL; *)
	hw_single_mode: Single;
	hw_cycle_mode: cycle;
	hw_cascade_mode: cascade;
	hw_mode_selector: Cascade_Cycle_Selector;
	hw_start_id_1: BOOL;
	hw_start_id_2: BOOL;
	info_analog_inputs_module: classInfoAnalogInputModule;
	hw_info_id_1: classInfoInvertorDrive;
	hw_info_id_2: classInfoInvertorDrive;
	ws_info_id_1: classInfoInvertorDrive;
	ws_info_id_2: classInfoInvertorDrive;
	hw_kpi_35: Kpi;
	hw_kpi_36: Kpi;
	ws_kpi_35: Kpi;
	ws_kpi_36: Kpi;
	plc_inputs: classPLC32m2StatusInputs;
	plc_outputs: classPLC32m2StatusOutputs;
	ws_single_mode: Single;
	ws_cycle_mode: cycle;
	ws_cascade_mode: cascade;
	ws_mode_selector: Cascade_Cycle_Selector;
	ws_start_id_1: BOOL;
	ws_start_id_2: BOOL;
	PLC_110_32_outputs: get_status_outputs;
	out_set_frequency: classParamsValueScaling;
	hw_mode_error: WORD;
	hw_alarm_manager: ALARM_MANAGER;
	(*hw_alarm_on: BOOL;
	ws_alarm_on: BOOL;*)
	ws_mode_error: WORD;
       hw_alarm_message AT %QW8.51.0: STRING(79);
       ws_alarm_message AT %QW8.91.0: STRING(79);

	hw_external_alarm: external_alarm_invertor_drive;
	ws_external_alarm: external_alarm_invertor_drive;
END_VAR

VAR RETAIN
	hw_settings_pressure_input: SetCurrentSensorPressure_4_20;
	hw_settings_pressure_output: SetCurrentSensorPressure_4_20;
	ws_settings_pressure_input: SetCurrentSensorPressure_4_20;
	ws_settings_pressure_output: SetCurrentSensorPressure_4_20;
END_VAR
VAR (* helpers for the ST form of the networks *)
	_t95 : REAL;
	_t97 : REAL;
	_t99 : REAL;
	_t83 : BOOL;
	_t84 : BOOL;
	_t85 : BOOL;
	_t204 : BOOL;
	_t205 : BOOL;
	_t206 : BOOL;
	_t207 : BOOL;
	_t277 : classParamsValueScaling;
	_t190 : REAL;
	_t191 : REAL;
	_t118 : BOOL;
	_t124 : BOOL;
	_t123 : BOOL;
	_t120 : BOOL;
	_t126 : BOOL;
	_t125 : BOOL;
	_t131 : BOOL;
	_t134 : BOOL;
	_t133 : BOOL;
	_t136 : BOOL;
	_t135 : BOOL;
	_t64 : TIME;
	_t65 : TIME;
	_t132 : BOOL;
	_t114 : TIME;
	_t115 : TIME;
	_t300 : BOOL;
	_t334 : BOOL;
END_VAR
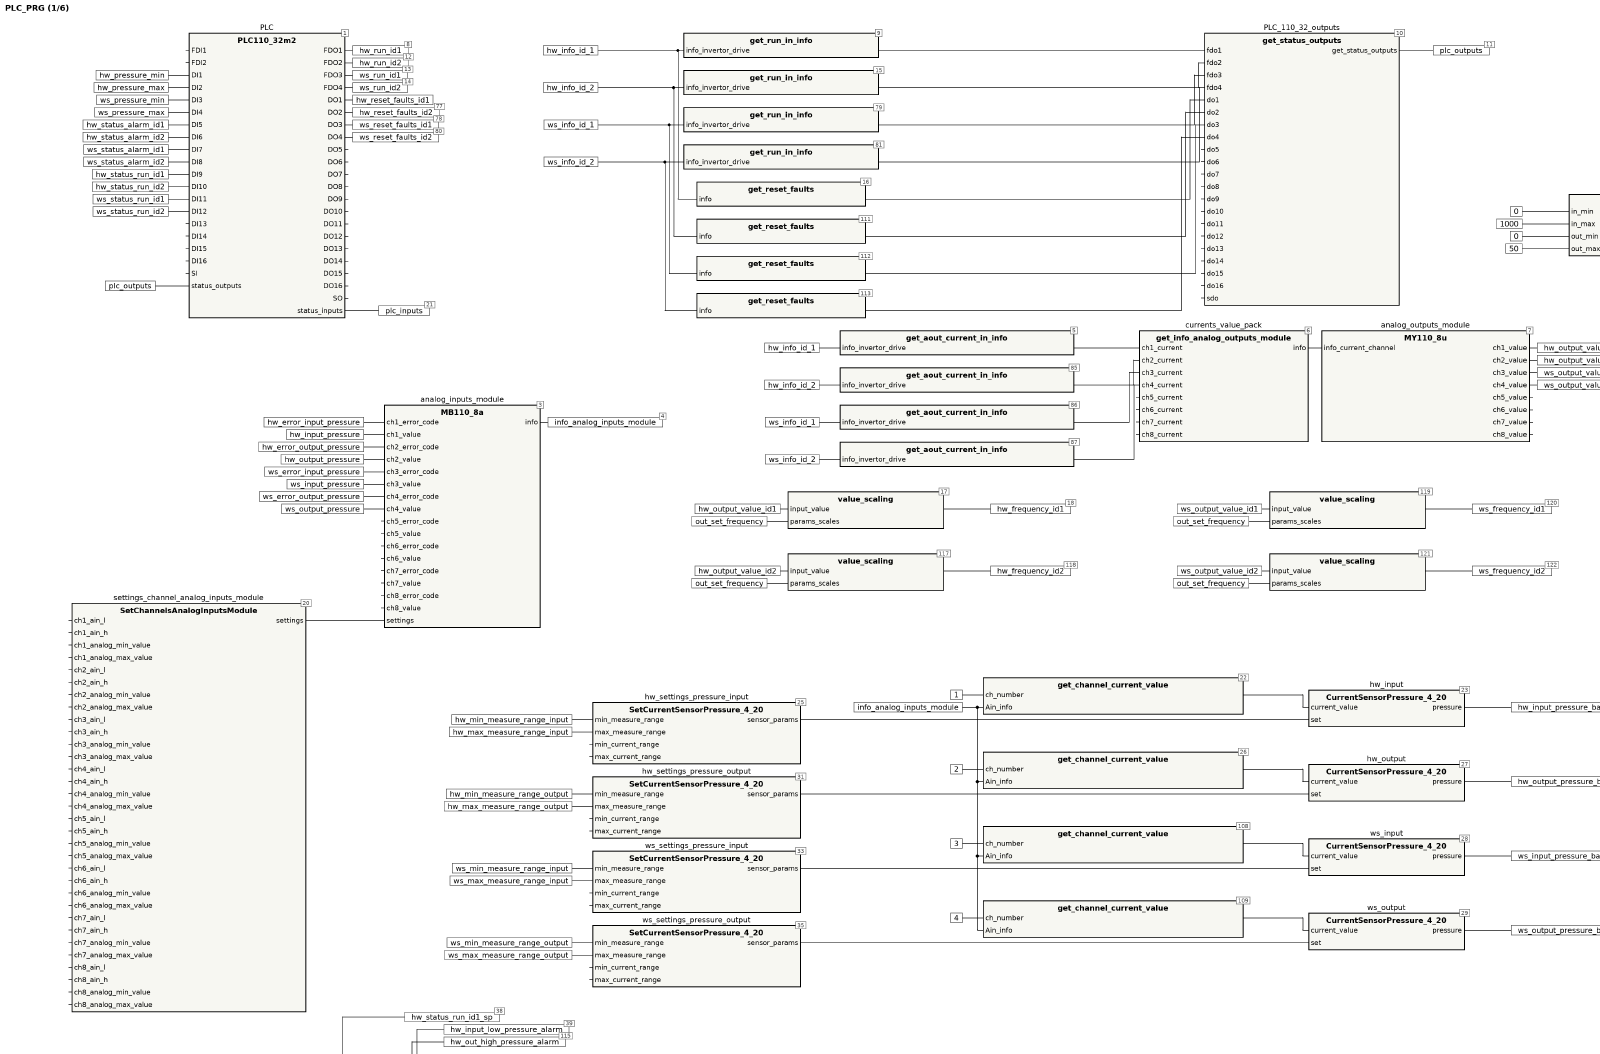
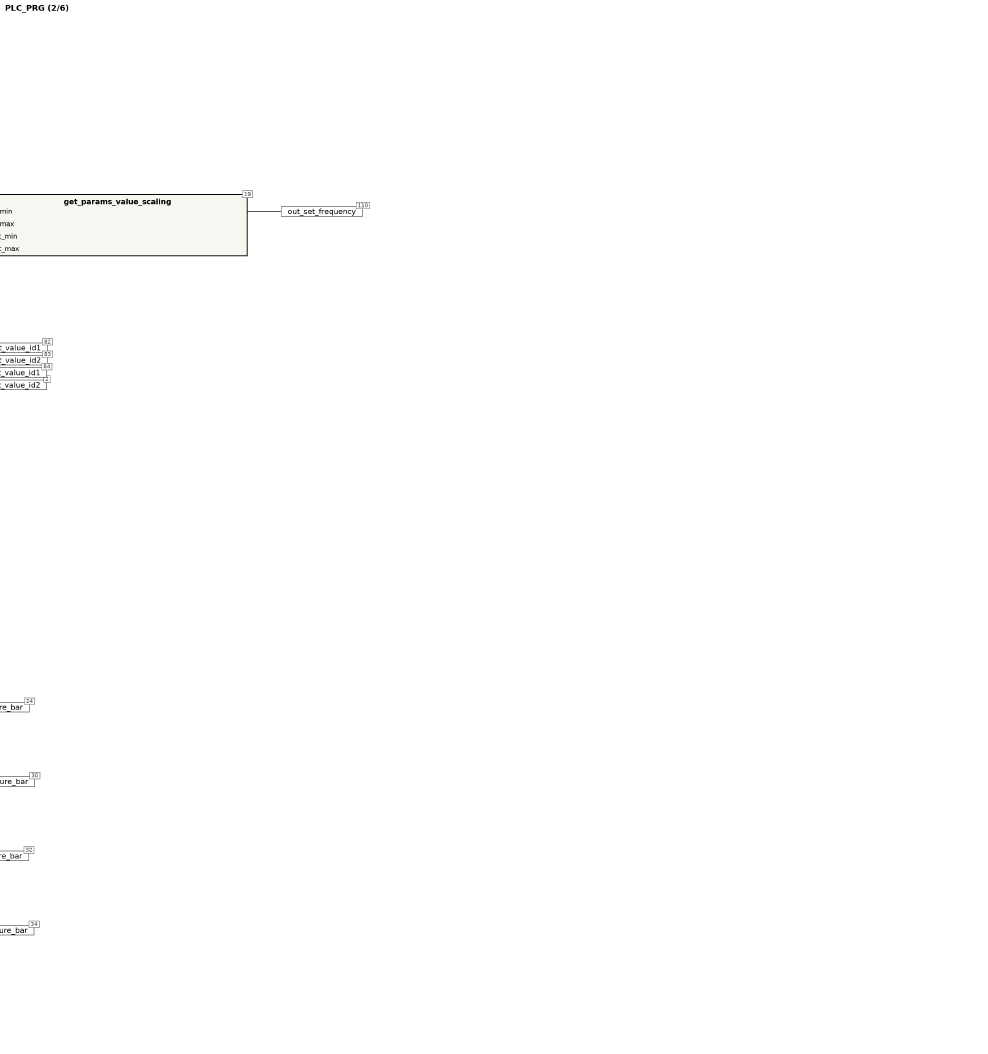
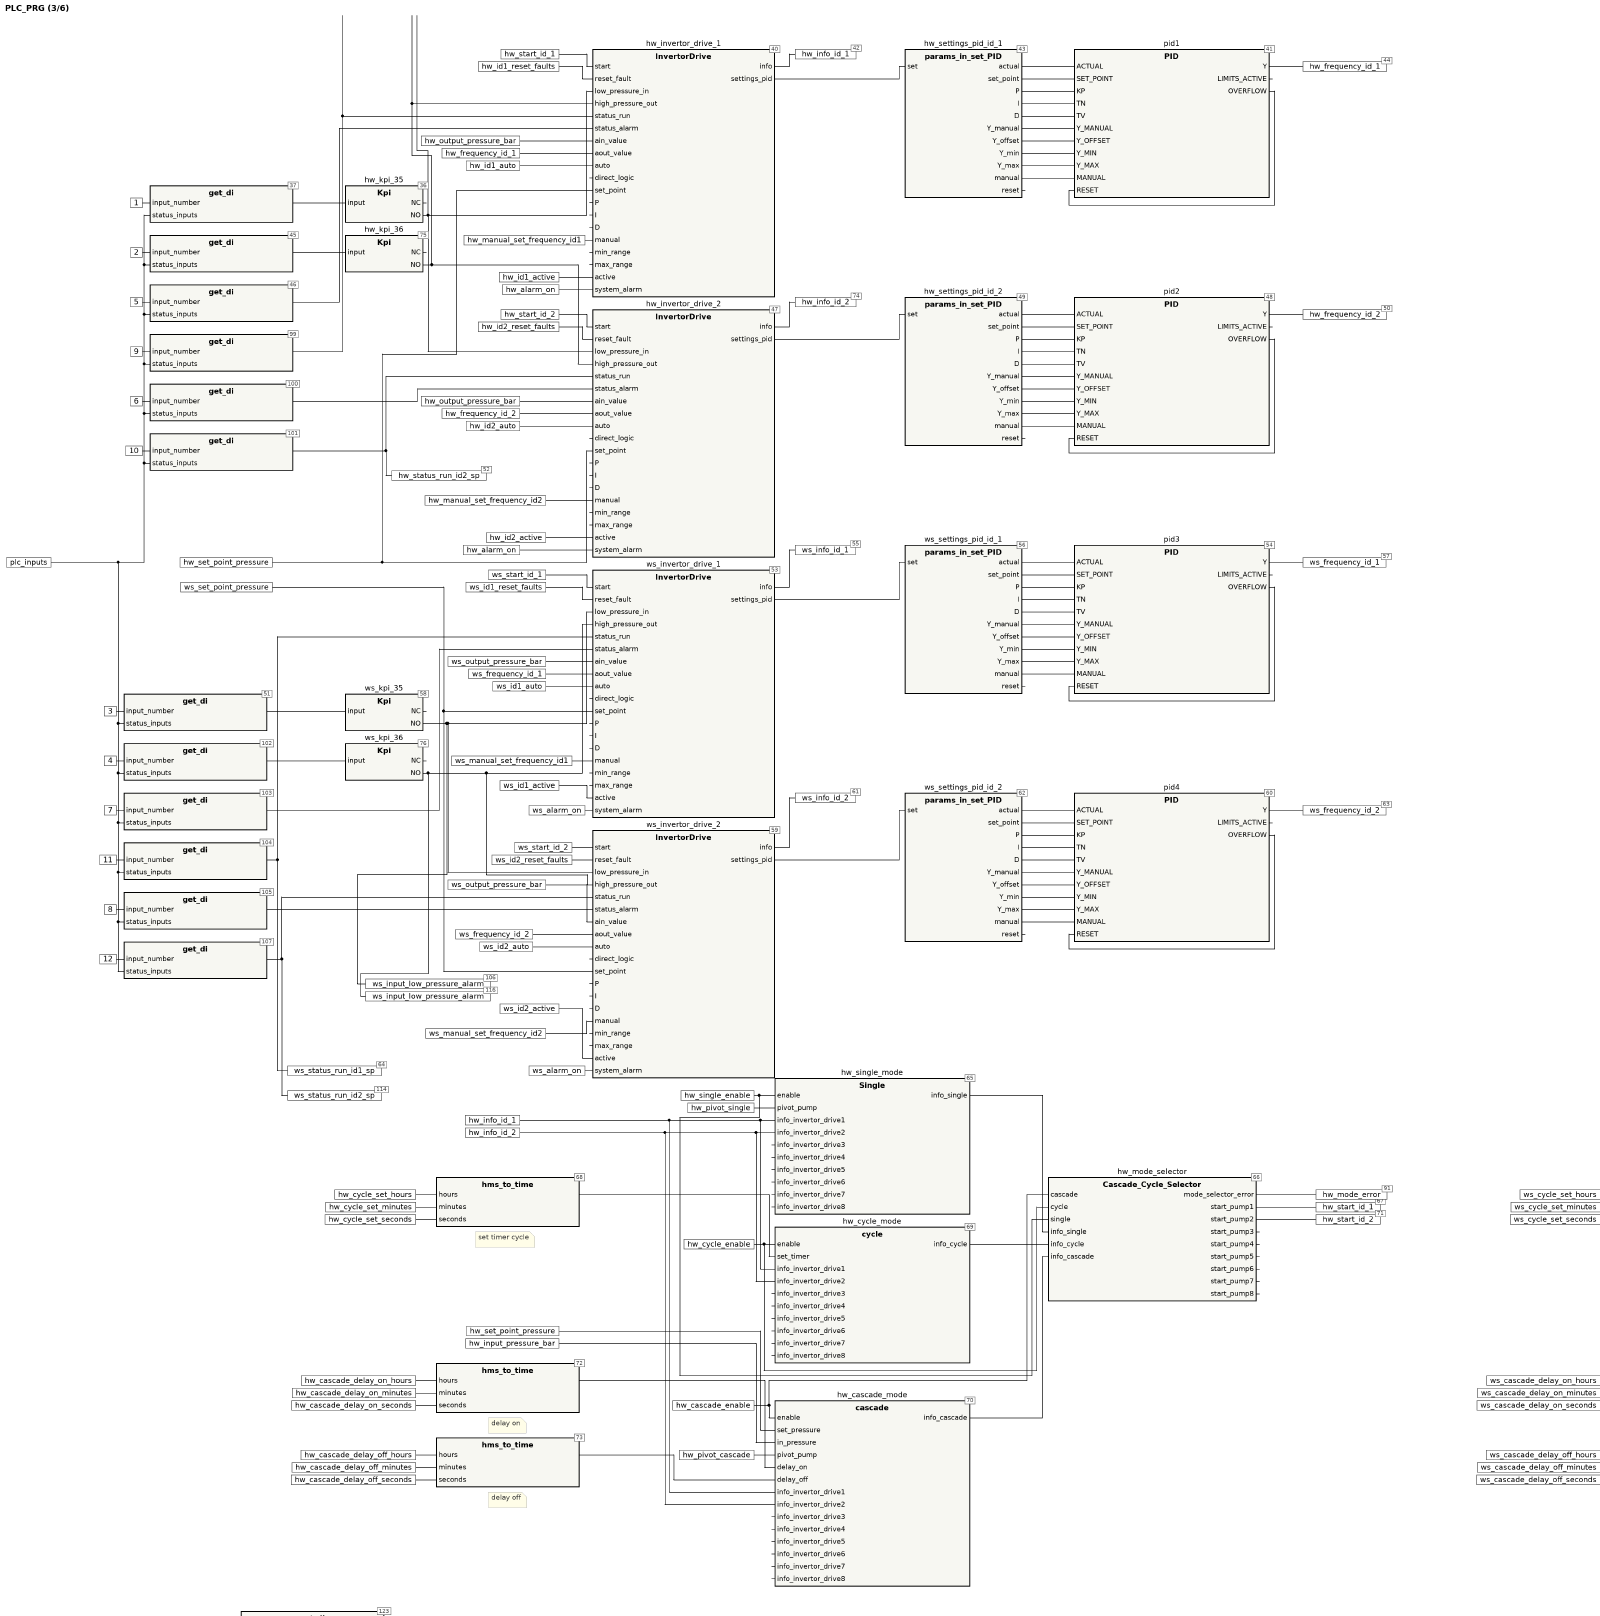
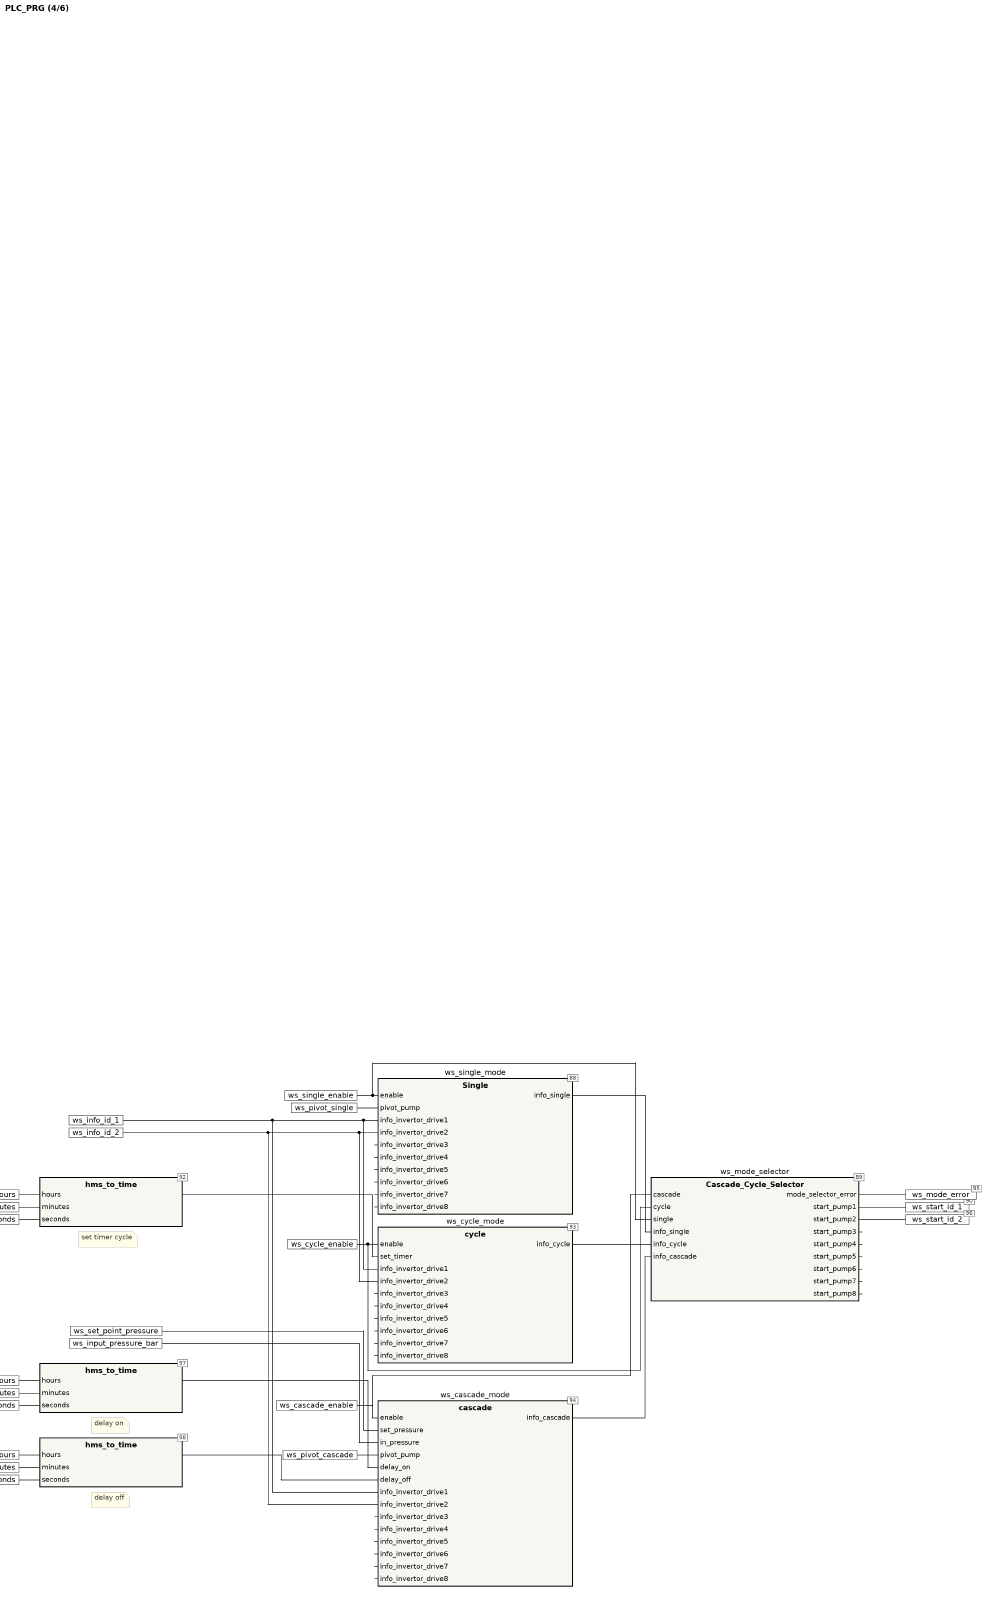
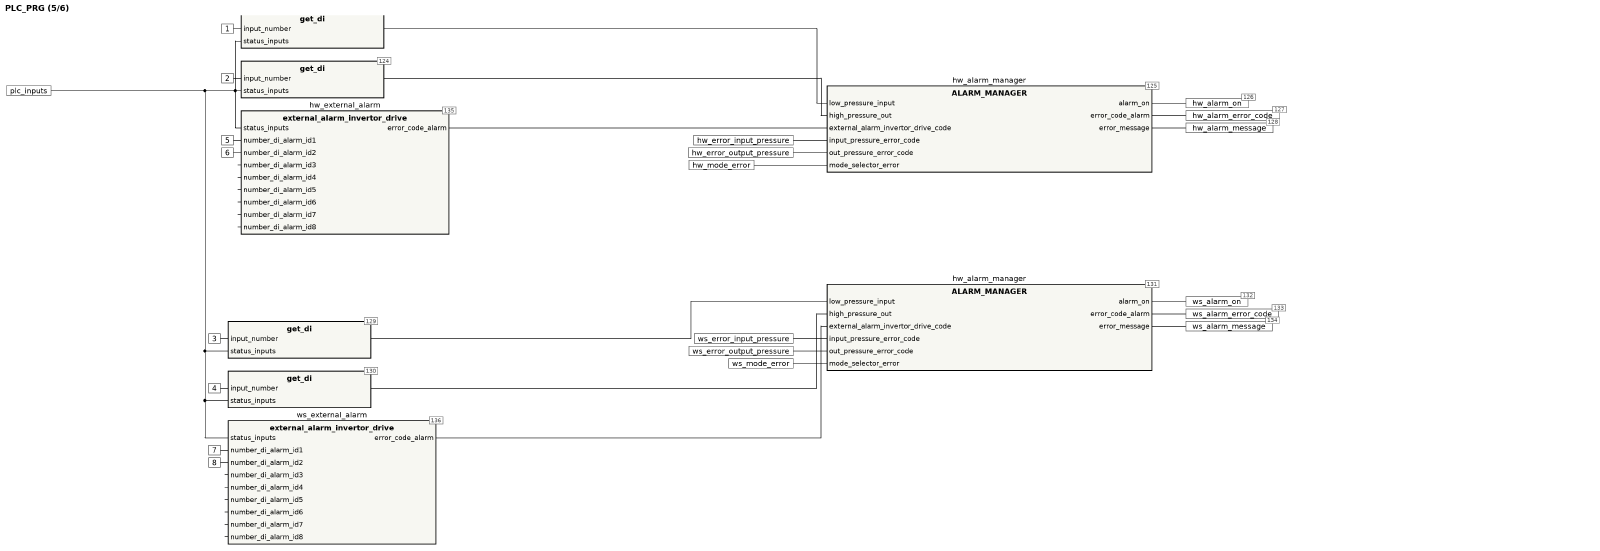
_CFC_ (* Continuous Function Chart, elements in execution order *)
(* set timer cycle *)
(* delay on *)
(* delay off *)
#0 hw_reset_faults_id1 <= #1.DO1
#1 PLC:PLC110_32m2(FDI1: -, FDI2: -, DI1: hw_pressure_min, DI2: hw_pressure_max, DI3: ws_pressure_min, DI4: ws_pressure_max, DI5: hw_status_alarm_id1, DI6: hw_status_alarm_id2, DI7: ws_status_alarm_id1, DI8: ws_status_alarm_id2, DI9: hw_status_run_id1, DI10: hw_status_run_id2, DI11: ws_status_run_id1, DI12: ws_status_run_id2, DI13: -, DI14: -, DI15: -, DI16: -, SI: -, status_outputs: plc_outputs)
#2 ws_output_value_id2 <= #7.ch4_value
#3 analog_inputs_module:MB110_8a(ch1_error_code: hw_error_input_pressure, ch1_value: hw_input_pressure, ch2_error_code: hw_error_output_pressure, ch2_value: hw_output_pressure, ch3_error_code: ws_error_input_pressure, ch3_value: ws_input_pressure, ch4_error_code: ws_error_output_pressure, ch4_value: ws_output_pressure, ch5_error_code: -, ch5_value: -, ch6_error_code: -, ch6_value: -, ch7_error_code: -, ch7_value: -, ch8_error_code: -, ch8_value: -, settings: #20.settings)
#4 info_analog_inputs_module <= #3.info
#5 get_aout_current_in_info(info_invertor_drive: hw_info_id_1)
#6 currents_value_pack:get_info_analog_outputs_module(ch1_current: #5, ch2_current: #85, ch3_current: #86, ch4_current: #87, ch5_current: -, ch6_current: -, ch7_current: -, ch8_current: -)
#7 analog_outputs_module:MY110_8u(info_current_channel: #6.info)
#8 hw_run_id1 <= #1.FDO1
#9 get_run_in_info(info_invertor_drive: hw_info_id_1)
#10 PLC_110_32_outputs:get_status_outputs(fdo1: #9, fdo2: #15, fdo3: #79, fdo4: #81, do1: #16, do2: #111, do3: #112, do4: #113, do5: -, do6: -, do7: -, do8: -, do9: -, do10: -, do11: -, do12: -, do13: -, do14: -, do15: -, do16: -, sdo: -)
#11 plc_outputs <= #10.get_status_outputs
#12 hw_run_id2 <= #1.FDO2
#13 ws_run_id1 <= #1.FDO3
#14 ws_run_id2 <= #1.FDO4
#15 get_run_in_info(info_invertor_drive: hw_info_id_2)
#16 get_reset_faults(info: hw_info_id_1)
#17 value_scaling(input_value: hw_output_value_id1, params_scales: out_set_frequency)
#18 hw_frequency_id1 <= #17
#19 get_params_value_scaling(in_min: 0, in_max: 1000, out_min: 0, out_max: 50)
#20 settings_channel_analog_inputs_module:SetChannelsAnalogInputsModule(ch1_ain_l: -, ch1_ain_h: -, ch1_analog_min_value: -, ch1_analog_max_value: -, ch2_ain_l: -, ch2_ain_h: -, ch2_analog_min_value: -, ch2_analog_max_value: -, ch3_ain_l: -, ch3_ain_h: -, ch3_analog_min_value: -, ch3_analog_max_value: -, ch4_ain_l: -, ch4_ain_h: -, ch4_analog_min_value: -, ch4_analog_max_value: -, ch5_ain_l: -, ch5_ain_h: -, ch5_analog_min_value: -, ch5_analog_max_value: -, ch6_ain_l: -, ch6_ain_h: -, ch6_analog_min_value: -, ch6_analog_max_value: -, ch7_ain_l: -, ch7_ain_h: -, ch7_analog_min_value: -, ch7_analog_max_value: -, ch8_ain_l: -, ch8_ain_h: -, ch8_analog_min_value: -, ch8_analog_max_value: -)
#21 plc_inputs <= #1.status_inputs
#22 get_channel_current_value(ch_number: 1, Ain_info: info_analog_inputs_module)
#23 hw_input:CurrentSensorPressure_4_20(current_value: #22, set: #25.sensor_params)
#24 hw_input_pressure_bar <= #23.pressure
#25 hw_settings_pressure_input:SetCurrentSensorPressure_4_20(min_measure_range: hw_min_measure_range_input, max_measure_range: hw_max_measure_range_input, min_current_range: -, max_current_range: -)
#26 get_channel_current_value(ch_number: 2, Ain_info: info_analog_inputs_module)
#27 hw_output:CurrentSensorPressure_4_20(current_value: #26, set: #31.sensor_params)
#28 ws_input:CurrentSensorPressure_4_20(current_value: #108, set: #33.sensor_params)
#29 ws_output:CurrentSensorPressure_4_20(current_value: #109, set: #35.sensor_params)
#30 hw_output_pressure_bar <= #27.pressure
#31 hw_settings_pressure_output:SetCurrentSensorPressure_4_20(min_measure_range: hw_min_measure_range_output, max_measure_range: hw_max_measure_range_output, min_current_range: -, max_current_range: -)
#32 ws_input_pressure_bar <= #28.pressure
#33 ws_settings_pressure_input:SetCurrentSensorPressure_4_20(min_measure_range: ws_min_measure_range_input, max_measure_range: ws_max_measure_range_input, min_current_range: -, max_current_range: -)
#34 ws_output_pressure_bar <= #29.pressure
#35 ws_settings_pressure_output:SetCurrentSensorPressure_4_20(min_measure_range: ws_min_measure_range_output, max_measure_range: ws_max_measure_range_output, min_current_range: -, max_current_range: -)
#36 hw_kpi_35:Kpi(input: #37)
#37 get_di(input_number: 1, status_inputs: plc_inputs)
#38 hw_status_run_id1_sp <= #99
#39 hw_input_low_pressure_alarm <= #36.NO
#40 hw_invertor_drive_1:InvertorDrive(start: hw_start_id_1, reset_fault: hw_id1_reset_faults, low_pressure_in: #36.NO, high_pressure_out: #75.NO, status_run: #99, status_alarm: #46, ain_value: hw_output_pressure_bar, aout_value: hw_frequency_id_1, auto: hw_id1_auto, direct_logic: -, set_point: hw_set_point_pressure, P: -, I: -, D: -, manual: hw_manual_set_frequency_id1, min_range: -, max_range: -, active: hw_id1_active, system_alarm: hw_alarm_on)
#41 pid1:PID(ACTUAL: #43.actual, SET_POINT: #43.set_point, KP: #43.P, TN: #43.I, TV: #43.D, Y_MANUAL: #43.Y_manual, Y_OFFSET: #43.Y_offset, Y_MIN: #43.Y_min, Y_MAX: #43.Y_max, MANUAL: #43.manual, RESET: #41.OVERFLOW)
#42 hw_info_id_1 <= #40.info
#43 hw_settings_pid_id_1:params_in_set_PID(set: #40.settings_pid)
#44 hw_frequency_id_1 <= #41.Y
#45 get_di(input_number: 2, status_inputs: plc_inputs)
#46 get_di(input_number: 5, status_inputs: plc_inputs)
#47 hw_invertor_drive_2:InvertorDrive(start: hw_start_id_2, reset_fault: hw_id2_reset_faults, low_pressure_in: #36.NO, high_pressure_out: #75.NO, status_run: #101, status_alarm: #100, ain_value: hw_output_pressure_bar, aout_value: hw_frequency_id_2, auto: hw_id2_auto, direct_logic: -, set_point: hw_set_point_pressure, P: -, I: -, D: -, manual: hw_manual_set_frequency_id2, min_range: -, max_range: -, active: hw_id2_active, system_alarm: hw_alarm_on)
#48 pid2:PID(ACTUAL: #49.actual, SET_POINT: #49.set_point, KP: #49.P, TN: #49.I, TV: #49.D, Y_MANUAL: #49.Y_manual, Y_OFFSET: #49.Y_offset, Y_MIN: #49.Y_min, Y_MAX: #49.Y_max, MANUAL: #49.manual, RESET: #48.OVERFLOW)
#49 hw_settings_pid_id_2:params_in_set_PID(set: #47.settings_pid)
#50 hw_frequency_id_2 <= #48.Y
#51 get_di(input_number: 3, status_inputs: plc_inputs)
#52 hw_status_run_id2_sp <= #101
#53 ws_invertor_drive_1:InvertorDrive(start: ws_start_id_1, reset_fault: ws_id1_reset_faults, low_pressure_in: #58.NO, high_pressure_out: #76.NO, status_run: #104, status_alarm: #103, ain_value: ws_output_pressure_bar, aout_value: ws_frequency_id_1, auto: ws_id1_auto, direct_logic: -, set_point: ws_set_point_pressure, P: -, I: -, D: -, manual: ws_manual_set_frequency_id1, min_range: -, max_range: -, active: ws_id1_active, system_alarm: ws_alarm_on)
#54 pid3:PID(ACTUAL: #56.actual, SET_POINT: #56.set_point, KP: #56.P, TN: #56.I, TV: #56.D, Y_MANUAL: #56.Y_manual, Y_OFFSET: #56.Y_offset, Y_MIN: #56.Y_min, Y_MAX: #56.Y_max, MANUAL: #56.manual, RESET: #54.OVERFLOW)
#55 ws_info_id_1 <= #53.info
#56 ws_settings_pid_id_1:params_in_set_PID(set: #53.settings_pid)
#57 ws_frequency_id_1 <= #54.Y
#58 ws_kpi_35:Kpi(input: #51)
#59 ws_invertor_drive_2:InvertorDrive(start: ws_start_id_2, reset_fault: ws_id2_reset_faults, low_pressure_in: #58.NO, high_pressure_out: #76.NO, status_run: #107, status_alarm: #105, ain_value: ws_output_pressure_bar, aout_value: ws_frequency_id_2, auto: ws_id2_auto, direct_logic: -, set_point: ws_set_point_pressure, P: -, I: -, D: -, manual: ws_manual_set_frequency_id2, min_range: -, max_range: -, active: ws_id2_active, system_alarm: ws_alarm_on)
#60 pid4:PID(ACTUAL: #62.actual, SET_POINT: #62.set_point, KP: #62.P, TN: #62.I, TV: #62.D, Y_MANUAL: #62.Y_manual, Y_OFFSET: #62.Y_offset, Y_MIN: #62.Y_min, Y_MAX: #62.Y_max, MANUAL: #62.manual, RESET: #60.OVERFLOW)
#61 ws_info_id_2 <= #59.info
#62 ws_settings_pid_id_2:params_in_set_PID(set: #59.settings_pid)
#63 ws_frequency_id_2 <= #60.Y
#64 ws_status_run_id1_sp <= #104
#65 hw_single_mode:Single(enable: hw_single_enable, pivot_pump: hw_pivot_single, info_invertor_drive1: hw_info_id_1, info_invertor_drive2: hw_info_id_2, info_invertor_drive3: -, info_invertor_drive4: -, info_invertor_drive5: -, info_invertor_drive6: -, info_invertor_drive7: -, info_invertor_drive8: -)
#66 hw_mode_selector:Cascade_Cycle_Selector(cascade: hw_cascade_enable, cycle: hw_cycle_enable, single: hw_single_enable, info_single: #65.info_single, info_cycle: #69.info_cycle, info_cascade: #70.info_cascade)
#67 hw_start_id_1 <= #66.start_pump1
#68 hms_to_time(hours: hw_cycle_set_hours, minutes: hw_cycle_set_minutes, seconds: hw_cycle_set_seconds)
#69 hw_cycle_mode:cycle(enable: hw_cycle_enable, set_timer: #68, info_invertor_drive1: hw_info_id_1, info_invertor_drive2: hw_info_id_2, info_invertor_drive3: -, info_invertor_drive4: -, info_invertor_drive5: -, info_invertor_drive6: -, info_invertor_drive7: -, info_invertor_drive8: -)
#70 hw_cascade_mode:cascade(enable: hw_cascade_enable, set_pressure: hw_set_point_pressure, in_pressure: hw_input_pressure_bar, pivot_pump: hw_pivot_cascade, delay_on: #72, delay_off: #73, info_invertor_drive1: hw_info_id_1, info_invertor_drive2: hw_info_id_2, info_invertor_drive3: -, info_invertor_drive4: -, info_invertor_drive5: -, info_invertor_drive6: -, info_invertor_drive7: -, info_invertor_drive8: -)
#71 hw_start_id_2 <= #66.start_pump2
#72 hms_to_time(hours: hw_cascade_delay_on_hours, minutes: hw_cascade_delay_on_minutes, seconds: hw_cascade_delay_on_seconds)
#73 hms_to_time(hours: hw_cascade_delay_off_hours, minutes: hw_cascade_delay_off_minutes, seconds: hw_cascade_delay_off_seconds)
#74 hw_info_id_2 <= #47.info
#75 hw_kpi_36:Kpi(input: #45)
#76 ws_kpi_36:Kpi(input: #102)
#77 hw_reset_faults_id2 <= #1.DO2
#78 ws_reset_faults_id1 <= #1.DO3
#79 get_run_in_info(info_invertor_drive: ws_info_id_1)
#80 ws_reset_faults_id2 <= #1.DO4
#81 get_run_in_info(info_invertor_drive: ws_info_id_2)
#82 hw_output_value_id1 <= #7.ch1_value
#83 hw_output_value_id2 <= #7.ch2_value
#84 ws_output_value_id1 <= #7.ch3_value
#85 get_aout_current_in_info(info_invertor_drive: hw_info_id_2)
#86 get_aout_current_in_info(info_invertor_drive: ws_info_id_1)
#87 get_aout_current_in_info(info_invertor_drive: ws_info_id_2)
(* set timer cycle *)
(* delay on *)
(* delay off *)
#88 ws_single_mode:Single(enable: ws_single_enable, pivot_pump: ws_pivot_single, info_invertor_drive1: ws_info_id_1, info_invertor_drive2: ws_info_id_2, info_invertor_drive3: -, info_invertor_drive4: -, info_invertor_drive5: -, info_invertor_drive6: -, info_invertor_drive7: -, info_invertor_drive8: -)
#89 ws_mode_selector:Cascade_Cycle_Selector(cascade: ws_cascade_enable, cycle: ws_cycle_enable, single: ws_single_enable, info_single: #88.info_single, info_cycle: #93.info_cycle, info_cascade: #94.info_cascade)
#90 ws_start_id_1 <= #89.start_pump1
#91 hw_mode_error <= #66.mode_selector_error
#92 hms_to_time(hours: ws_cycle_set_hours, minutes: ws_cycle_set_minutes, seconds: ws_cycle_set_seconds)
#93 ws_cycle_mode:cycle(enable: ws_cycle_enable, set_timer: #92, info_invertor_drive1: ws_info_id_1, info_invertor_drive2: ws_info_id_2, info_invertor_drive3: -, info_invertor_drive4: -, info_invertor_drive5: -, info_invertor_drive6: -, info_invertor_drive7: -, info_invertor_drive8: -)
#94 ws_cascade_mode:cascade(enable: ws_cascade_enable, set_pressure: ws_set_point_pressure, in_pressure: ws_input_pressure_bar, pivot_pump: ws_pivot_cascade, delay_on: #97, delay_off: #98, info_invertor_drive1: ws_info_id_1, info_invertor_drive2: ws_info_id_2, info_invertor_drive3: -, info_invertor_drive4: -, info_invertor_drive5: -, info_invertor_drive6: -, info_invertor_drive7: -, info_invertor_drive8: -)
#95 ws_mode_error <= #89.mode_selector_error
#96 ws_start_id_2 <= #89.start_pump2
#97 hms_to_time(hours: ws_cascade_delay_on_hours, minutes: ws_cascade_delay_on_minutes, seconds: ws_cascade_delay_on_seconds)
#98 hms_to_time(hours: ws_cascade_delay_off_hours, minutes: ws_cascade_delay_off_minutes, seconds: ws_cascade_delay_off_seconds)
#99 get_di(input_number: 9, status_inputs: plc_inputs)
#100 get_di(input_number: 6, status_inputs: plc_inputs)
#101 get_di(input_number: 10, status_inputs: plc_inputs)
#102 get_di(input_number: 4, status_inputs: plc_inputs)
#103 get_di(input_number: 7, status_inputs: plc_inputs)
#104 get_di(input_number: 11, status_inputs: plc_inputs)
#105 get_di(input_number: 8, status_inputs: plc_inputs)
#106 ws_input_low_pressure_alarm <= #58.NO
#107 get_di(input_number: 12, status_inputs: plc_inputs)
#108 get_channel_current_value(ch_number: 3, Ain_info: info_analog_inputs_module)
#109 get_channel_current_value(ch_number: 4, Ain_info: info_analog_inputs_module)
#110 out_set_frequency <= #19
#111 get_reset_faults(info: hw_info_id_2)
#112 get_reset_faults(info: ws_info_id_1)
#113 get_reset_faults(info: ws_info_id_2)
#114 ws_status_run_id2_sp <= #107
#115 hw_out_high_pressure_alarm <= #75.NO
#116 ws_input_low_pressure_alarm <= #76.NO
#117 value_scaling(input_value: hw_output_value_id2, params_scales: out_set_frequency)
#118 hw_frequency_id2 <= #117
#119 value_scaling(input_value: ws_output_value_id1, params_scales: out_set_frequency)
#120 ws_frequency_id1 <= #119
#121 value_scaling(input_value: ws_output_value_id2, params_scales: out_set_frequency)
#122 ws_frequency_id2 <= #121
#123 get_di(input_number: 1, status_inputs: plc_inputs)
#124 get_di(input_number: 2, status_inputs: plc_inputs)
#125 hw_alarm_manager:ALARM_MANAGER(low_pressure_input: #123, high_pressure_out: #124, external_alarm_invertor_drive_code: #135.error_code_alarm, input_pressure_error_code: hw_error_input_pressure, out_pressure_error_code: hw_error_output_pressure, mode_selector_error: hw_mode_error)
#126 hw_alarm_on <= #125.alarm_on
#127 hw_alarm_error_code <= #125.error_code_alarm
#128 hw_alarm_message <= #125.error_message
#129 get_di(input_number: 3, status_inputs: plc_inputs)
#130 get_di(input_number: 4, status_inputs: plc_inputs)
#131 hw_alarm_manager:ALARM_MANAGER(low_pressure_input: #129, high_pressure_out: #130, external_alarm_invertor_drive_code: #136.error_code_alarm, input_pressure_error_code: ws_error_input_pressure, out_pressure_error_code: ws_error_output_pressure, mode_selector_error: ws_mode_error)
#132 ws_alarm_on <= #131.alarm_on
#133 ws_alarm_error_code <= #131.error_code_alarm
#134 ws_alarm_message <= #131.error_message
#135 hw_external_alarm:external_alarm_invertor_drive(status_inputs: plc_inputs, number_di_alarm_id1: 5, number_di_alarm_id2: 6, number_di_alarm_id3: -, number_di_alarm_id4: -, number_di_alarm_id5: -, number_di_alarm_id6: -, number_di_alarm_id7: -, number_di_alarm_id8: -)
#136 ws_external_alarm:external_alarm_invertor_drive(status_inputs: plc_inputs, number_di_alarm_id1: 7, number_di_alarm_id2: 8, number_di_alarm_id3: -, number_di_alarm_id4: -, number_di_alarm_id5: -, number_di_alarm_id6: -, number_di_alarm_id7: -, number_di_alarm_id8: -)
_END_CFC_
(* the same logic as Structured Text *)
(* set timer cycle *)
(* delay on *)
(* delay off *)
hw_reset_faults_id1 := PLC.DO1;
PLC(DI1 := hw_pressure_min, DI2 := hw_pressure_max, DI3 := ws_pressure_min, DI4 := ws_pressure_max, DI5 := hw_status_alarm_id1, DI6 := hw_status_alarm_id2, DI7 := ws_status_alarm_id1, DI8 := ws_status_alarm_id2, DI9 := hw_status_run_id1, DI10 := hw_status_run_id2, DI11 := ws_status_run_id1, DI12 := ws_status_run_id2, status_outputs := plc_outputs);
ws_output_value_id2 := analog_outputs_module.ch4_value;
analog_inputs_module(ch1_error_code := hw_error_input_pressure, ch1_value := hw_input_pressure, ch2_error_code := hw_error_output_pressure, ch2_value := hw_output_pressure, ch3_error_code := ws_error_input_pressure, ch3_value := ws_input_pressure, ch4_error_code := ws_error_output_pressure, ch4_value := ws_output_pressure, settings := settings_channel_analog_inputs_module.settings);
info_analog_inputs_module := analog_inputs_module.info;
currents_value_pack(ch1_current := get_aout_current_in_info(info_invertor_drive := hw_info_id_1), ch2_current := _t95, ch3_current := _t97, ch4_current := _t99);
analog_outputs_module(info_current_channel := currents_value_pack.info);
hw_run_id1 := PLC.FDO1;
PLC_110_32_outputs(fdo1 := get_run_in_info(info_invertor_drive := hw_info_id_1), fdo2 := _t83, fdo3 := _t84, fdo4 := _t85, do1 := _t204, do2 := _t205, do3 := _t206, do4 := _t207);
plc_outputs := PLC_110_32_outputs.get_status_outputs;
hw_run_id2 := PLC.FDO2;
ws_run_id1 := PLC.FDO3;
ws_run_id2 := PLC.FDO4;
_t83 := get_run_in_info(info_invertor_drive := hw_info_id_2);
_t204 := get_reset_faults(info := hw_info_id_1);
hw_frequency_id1 := value_scaling(input_value := hw_output_value_id1, params_scales := out_set_frequency);
_t277 := get_params_value_scaling(in_min := 0, in_max := 1000, out_min := 0, out_max := 50);
settings_channel_analog_inputs_module();
plc_inputs := PLC.status_inputs;
hw_input(current_value := get_channel_current_value(ch_number := 1, Ain_info := info_analog_inputs_module), set := hw_settings_pressure_input.sensor_params);
hw_input_pressure_bar := hw_input.pressure;
hw_settings_pressure_input(min_measure_range := hw_min_measure_range_input, max_measure_range := hw_max_measure_range_input);
hw_output(current_value := get_channel_current_value(ch_number := 2, Ain_info := info_analog_inputs_module), set := hw_settings_pressure_output.sensor_params);
ws_input(current_value := _t190, set := ws_settings_pressure_input.sensor_params);
ws_output(current_value := _t191, set := ws_settings_pressure_output.sensor_params);
hw_output_pressure_bar := hw_output.pressure;
hw_settings_pressure_output(min_measure_range := hw_min_measure_range_output, max_measure_range := hw_max_measure_range_output);
ws_input_pressure_bar := ws_input.pressure;
ws_settings_pressure_input(min_measure_range := ws_min_measure_range_input, max_measure_range := ws_max_measure_range_input);
ws_output_pressure_bar := ws_output.pressure;
ws_settings_pressure_output(min_measure_range := ws_min_measure_range_output, max_measure_range := ws_max_measure_range_output);
hw_kpi_35(input := _t118);
_t118 := get_di(input_number := 1, status_inputs := plc_inputs);
hw_status_run_id1_sp := _t124;
hw_input_low_pressure_alarm := hw_kpi_35.NO;
hw_invertor_drive_1(start := hw_start_id_1, reset_fault := hw_id1_reset_faults, low_pressure_in := hw_kpi_35.NO, high_pressure_out := hw_kpi_36.NO, status_run := _t124, status_alarm := _t123, ain_value := hw_output_pressure_bar, aout_value := hw_frequency_id_1, auto := hw_id1_auto, set_point := hw_set_point_pressure, manual := hw_manual_set_frequency_id1, active := hw_id1_active, system_alarm := hw_alarm_on);
pid1(ACTUAL := hw_settings_pid_id_1.actual, SET_POINT := hw_settings_pid_id_1.set_point, KP := hw_settings_pid_id_1.P, TN := hw_settings_pid_id_1.I, TV := hw_settings_pid_id_1.D, Y_MANUAL := hw_settings_pid_id_1.Y_manual, Y_OFFSET := hw_settings_pid_id_1.Y_offset, Y_MIN := hw_settings_pid_id_1.Y_min, Y_MAX := hw_settings_pid_id_1.Y_max, MANUAL := hw_settings_pid_id_1.manual, RESET := pid1.OVERFLOW);
hw_info_id_1 := hw_invertor_drive_1.info;
hw_settings_pid_id_1(set := hw_invertor_drive_1.settings_pid);
hw_frequency_id_1 := pid1.Y;
_t120 := get_di(input_number := 2, status_inputs := plc_inputs);
_t123 := get_di(input_number := 5, status_inputs := plc_inputs);
hw_invertor_drive_2(start := hw_start_id_2, reset_fault := hw_id2_reset_faults, low_pressure_in := hw_kpi_35.NO, high_pressure_out := hw_kpi_36.NO, status_run := _t126, status_alarm := _t125, ain_value := hw_output_pressure_bar, aout_value := hw_frequency_id_2, auto := hw_id2_auto, set_point := hw_set_point_pressure, manual := hw_manual_set_frequency_id2, active := hw_id2_active, system_alarm := hw_alarm_on);
pid2(ACTUAL := hw_settings_pid_id_2.actual, SET_POINT := hw_settings_pid_id_2.set_point, KP := hw_settings_pid_id_2.P, TN := hw_settings_pid_id_2.I, TV := hw_settings_pid_id_2.D, Y_MANUAL := hw_settings_pid_id_2.Y_manual, Y_OFFSET := hw_settings_pid_id_2.Y_offset, Y_MIN := hw_settings_pid_id_2.Y_min, Y_MAX := hw_settings_pid_id_2.Y_max, MANUAL := hw_settings_pid_id_2.manual, RESET := pid2.OVERFLOW);
hw_settings_pid_id_2(set := hw_invertor_drive_2.settings_pid);
hw_frequency_id_2 := pid2.Y;
_t131 := get_di(input_number := 3, status_inputs := plc_inputs);
hw_status_run_id2_sp := _t126;
ws_invertor_drive_1(start := ws_start_id_1, reset_fault := ws_id1_reset_faults, low_pressure_in := ws_kpi_35.NO, high_pressure_out := ws_kpi_36.NO, status_run := _t134, status_alarm := _t133, ain_value := ws_output_pressure_bar, aout_value := ws_frequency_id_1, auto := ws_id1_auto, set_point := ws_set_point_pressure, manual := ws_manual_set_frequency_id1, active := ws_id1_active, system_alarm := ws_alarm_on);
pid3(ACTUAL := ws_settings_pid_id_1.actual, SET_POINT := ws_settings_pid_id_1.set_point, KP := ws_settings_pid_id_1.P, TN := ws_settings_pid_id_1.I, TV := ws_settings_pid_id_1.D, Y_MANUAL := ws_settings_pid_id_1.Y_manual, Y_OFFSET := ws_settings_pid_id_1.Y_offset, Y_MIN := ws_settings_pid_id_1.Y_min, Y_MAX := ws_settings_pid_id_1.Y_max, MANUAL := ws_settings_pid_id_1.manual, RESET := pid3.OVERFLOW);
ws_info_id_1 := ws_invertor_drive_1.info;
ws_settings_pid_id_1(set := ws_invertor_drive_1.settings_pid);
ws_frequency_id_1 := pid3.Y;
ws_kpi_35(input := _t131);
ws_invertor_drive_2(start := ws_start_id_2, reset_fault := ws_id2_reset_faults, low_pressure_in := ws_kpi_35.NO, high_pressure_out := ws_kpi_36.NO, status_run := _t136, status_alarm := _t135, ain_value := ws_output_pressure_bar, aout_value := ws_frequency_id_2, auto := ws_id2_auto, set_point := ws_set_point_pressure, manual := ws_manual_set_frequency_id2, active := ws_id2_active, system_alarm := ws_alarm_on);
pid4(ACTUAL := ws_settings_pid_id_2.actual, SET_POINT := ws_settings_pid_id_2.set_point, KP := ws_settings_pid_id_2.P, TN := ws_settings_pid_id_2.I, TV := ws_settings_pid_id_2.D, Y_MANUAL := ws_settings_pid_id_2.Y_manual, Y_OFFSET := ws_settings_pid_id_2.Y_offset, Y_MIN := ws_settings_pid_id_2.Y_min, Y_MAX := ws_settings_pid_id_2.Y_max, MANUAL := ws_settings_pid_id_2.manual, RESET := pid4.OVERFLOW);
ws_info_id_2 := ws_invertor_drive_2.info;
ws_settings_pid_id_2(set := ws_invertor_drive_2.settings_pid);
ws_frequency_id_2 := pid4.Y;
ws_status_run_id1_sp := _t134;
hw_single_mode(enable := hw_single_enable, pivot_pump := hw_pivot_single, info_invertor_drive1 := hw_info_id_1, info_invertor_drive2 := hw_info_id_2);
hw_mode_selector(cascade := hw_cascade_enable, cycle := hw_cycle_enable, single := hw_single_enable, info_single := hw_single_mode.info_single, info_cycle := hw_cycle_mode.info_cycle, info_cascade := hw_cascade_mode.info_cascade);
hw_start_id_1 := hw_mode_selector.start_pump1;
hw_cycle_mode(enable := hw_cycle_enable, set_timer := hms_to_time(hours := hw_cycle_set_hours, minutes := hw_cycle_set_minutes, seconds := hw_cycle_set_seconds), info_invertor_drive1 := hw_info_id_1, info_invertor_drive2 := hw_info_id_2);
hw_cascade_mode(enable := hw_cascade_enable, set_pressure := hw_set_point_pressure, in_pressure := hw_input_pressure_bar, pivot_pump := hw_pivot_cascade, delay_on := _t64, delay_off := _t65, info_invertor_drive1 := hw_info_id_1, info_invertor_drive2 := hw_info_id_2);
hw_start_id_2 := hw_mode_selector.start_pump2;
_t64 := hms_to_time(hours := hw_cascade_delay_on_hours, minutes := hw_cascade_delay_on_minutes, seconds := hw_cascade_delay_on_seconds);
_t65 := hms_to_time(hours := hw_cascade_delay_off_hours, minutes := hw_cascade_delay_off_minutes, seconds := hw_cascade_delay_off_seconds);
hw_info_id_2 := hw_invertor_drive_2.info;
hw_kpi_36(input := _t120);
ws_kpi_36(input := _t132);
hw_reset_faults_id2 := PLC.DO2;
ws_reset_faults_id1 := PLC.DO3;
_t84 := get_run_in_info(info_invertor_drive := ws_info_id_1);
ws_reset_faults_id2 := PLC.DO4;
_t85 := get_run_in_info(info_invertor_drive := ws_info_id_2);
hw_output_value_id1 := analog_outputs_module.ch1_value;
hw_output_value_id2 := analog_outputs_module.ch2_value;
ws_output_value_id1 := analog_outputs_module.ch3_value;
_t95 := get_aout_current_in_info(info_invertor_drive := hw_info_id_2);
_t97 := get_aout_current_in_info(info_invertor_drive := ws_info_id_1);
_t99 := get_aout_current_in_info(info_invertor_drive := ws_info_id_2);
(* set timer cycle *)
(* delay on *)
(* delay off *)
ws_single_mode(enable := ws_single_enable, pivot_pump := ws_pivot_single, info_invertor_drive1 := ws_info_id_1, info_invertor_drive2 := ws_info_id_2);
ws_mode_selector(cascade := ws_cascade_enable, cycle := ws_cycle_enable, single := ws_single_enable, info_single := ws_single_mode.info_single, info_cycle := ws_cycle_mode.info_cycle, info_cascade := ws_cascade_mode.info_cascade);
ws_start_id_1 := ws_mode_selector.start_pump1;
hw_mode_error := hw_mode_selector.mode_selector_error;
ws_cycle_mode(enable := ws_cycle_enable, set_timer := hms_to_time(hours := ws_cycle_set_hours, minutes := ws_cycle_set_minutes, seconds := ws_cycle_set_seconds), info_invertor_drive1 := ws_info_id_1, info_invertor_drive2 := ws_info_id_2);
ws_cascade_mode(enable := ws_cascade_enable, set_pressure := ws_set_point_pressure, in_pressure := ws_input_pressure_bar, pivot_pump := ws_pivot_cascade, delay_on := _t114, delay_off := _t115, info_invertor_drive1 := ws_info_id_1, info_invertor_drive2 := ws_info_id_2);
ws_mode_error := ws_mode_selector.mode_selector_error;
ws_start_id_2 := ws_mode_selector.start_pump2;
_t114 := hms_to_time(hours := ws_cascade_delay_on_hours, minutes := ws_cascade_delay_on_minutes, seconds := ws_cascade_delay_on_seconds);
_t115 := hms_to_time(hours := ws_cascade_delay_off_hours, minutes := ws_cascade_delay_off_minutes, seconds := ws_cascade_delay_off_seconds);
_t124 := get_di(input_number := 9, status_inputs := plc_inputs);
_t125 := get_di(input_number := 6, status_inputs := plc_inputs);
_t126 := get_di(input_number := 10, status_inputs := plc_inputs);
_t132 := get_di(input_number := 4, status_inputs := plc_inputs);
_t133 := get_di(input_number := 7, status_inputs := plc_inputs);
_t134 := get_di(input_number := 11, status_inputs := plc_inputs);
_t135 := get_di(input_number := 8, status_inputs := plc_inputs);
ws_input_low_pressure_alarm := ws_kpi_35.NO;
_t136 := get_di(input_number := 12, status_inputs := plc_inputs);
_t190 := get_channel_current_value(ch_number := 3, Ain_info := info_analog_inputs_module);
_t191 := get_channel_current_value(ch_number := 4, Ain_info := info_analog_inputs_module);
out_set_frequency := _t277;
_t205 := get_reset_faults(info := hw_info_id_2);
_t206 := get_reset_faults(info := ws_info_id_1);
_t207 := get_reset_faults(info := ws_info_id_2);
ws_status_run_id2_sp := _t136;
hw_out_high_pressure_alarm := hw_kpi_36.NO;
ws_input_low_pressure_alarm := ws_kpi_36.NO;
hw_frequency_id2 := value_scaling(input_value := hw_output_value_id2, params_scales := out_set_frequency);
ws_frequency_id1 := value_scaling(input_value := ws_output_value_id1, params_scales := out_set_frequency);
ws_frequency_id2 := value_scaling(input_value := ws_output_value_id2, params_scales := out_set_frequency);
_t300 := get_di(input_number := 1, status_inputs := plc_inputs);
hw_alarm_manager(low_pressure_input := _t300, high_pressure_out := get_di(input_number := 2, status_inputs := plc_inputs), external_alarm_invertor_drive_code := hw_external_alarm.error_code_alarm, input_pressure_error_code := hw_error_input_pressure, out_pressure_error_code := hw_error_output_pressure, mode_selector_error := hw_mode_error);
hw_alarm_on := hw_alarm_manager.alarm_on;
hw_alarm_error_code := hw_alarm_manager.error_code_alarm;
hw_alarm_message := hw_alarm_manager.error_message;
_t334 := get_di(input_number := 3, status_inputs := plc_inputs);
hw_alarm_manager(low_pressure_input := _t334, high_pressure_out := get_di(input_number := 4, status_inputs := plc_inputs), external_alarm_invertor_drive_code := ws_external_alarm.error_code_alarm, input_pressure_error_code := ws_error_input_pressure, out_pressure_error_code := ws_error_output_pressure, mode_selector_error := ws_mode_error);
ws_alarm_on := hw_alarm_manager.alarm_on;
ws_alarm_error_code := hw_alarm_manager.error_code_alarm;
ws_alarm_message := hw_alarm_manager.error_message;
hw_external_alarm(status_inputs := plc_inputs, number_di_alarm_id1 := 5, number_di_alarm_id2 := 6);
ws_external_alarm(status_inputs := plc_inputs, number_di_alarm_id1 := 7, number_di_alarm_id2 := 8);
END_PROGRAM

(* POU PLC110_32/PLC110_32m2, ST *)
FUNCTION_BLOCK PLC110_32m2

VAR_INPUT
	FDI1:BOOL;
	FDI2:BOOL;
	DI1:BOOL;
	DI2:BOOL;
	DI3:BOOL;
	DI4:BOOL;
	DI5:BOOL;
	DI6:BOOL;
	DI7:BOOL;
	DI8:BOOL;
	DI9:BOOL;
	DI10:BOOL;
	DI11:BOOL;
	DI12:BOOL;
	DI13:BOOL;
	DI14:BOOL;
	DI15:BOOL;
	DI16:BOOL;
	SI:BOOL;
	status_outputs:classPLC32m2StatusOutputs;
END_VAR

VAR_OUTPUT
	FDO1:BOOL;
	FDO2:BOOL;
	FDO3:BOOL;
	FDO4:BOOL;
	DO1:BOOL;
	DO2:BOOL;
	DO3:BOOL;
	DO4:BOOL;
	DO5:BOOL;
	DO6:BOOL;
	DO7:BOOL;
	DO8:BOOL;
	DO9:BOOL;
	DO10:BOOL;
	DO11:BOOL;
	DO12:BOOL;
	DO13:BOOL;
	DO14:BOOL;
	DO15:BOOL;
	DO16:BOOL;
	SO:BOOL;
	status_inputs:classPLC32m2StatusInputs;
END_VAR

VAR
	fast_inputs:classFastDiscreteInputs;
	discrete_inputs:classDiscreteInputs;
	special_input:classSpecialInput;
	fast_outputs:classFastDiscreteOutputs;
	discrete_outputs:classDiscreteOutputs;
	special_output:classSpecialOutput;
END_VAR
init;

get_status_inputs;

get_status_outputs;
END_FUNCTION_BLOCK
ACTION get_status_inputs:
status_inputs.fast_inputs:=fast_inputs;
status_inputs.discrete_inputs:=discrete_inputs;
status_inputs.special_input:=special_input;
END_ACTION
ACTION get_status_outputs:
FDO1:=status_outputs.fast_outputs.Bit1;
FDO2:=status_outputs.fast_outputs.Bit2;
FDO3:=status_outputs.fast_outputs.Bit3;
FDO4:=status_outputs.fast_outputs.Bit4;

DO1:=status_outputs.discrete_outputs.first_byte.Bit1;
DO2:=status_outputs.discrete_outputs.first_byte.Bit2;
DO3:=status_outputs.discrete_outputs.first_byte.Bit3;
DO4:=status_outputs.discrete_outputs.first_byte.Bit4;
DO5:=status_outputs.discrete_outputs.first_byte.Bit5;
DO6:=status_outputs.discrete_outputs.first_byte.Bit6;
DO7:=status_outputs.discrete_outputs.first_byte.Bit7;
DO8:=status_outputs.discrete_outputs.first_byte.Bit8;
DO9:=status_outputs.discrete_outputs.second_byte.Bit1;
DO10:=status_outputs.discrete_outputs.second_byte.Bit2;
DO11:=status_outputs.discrete_outputs.second_byte.Bit3;
DO12:=status_outputs.discrete_outputs.second_byte.Bit4;
DO13:=status_outputs.discrete_outputs.second_byte.Bit5;
DO14:=status_outputs.discrete_outputs.second_byte.Bit6;
DO15:=status_outputs.discrete_outputs.second_byte.Bit7;
DO16:=status_outputs.discrete_outputs.second_byte.Bit8;

SO:=status_outputs.special_output.Bit1;
END_ACTION
ACTION init:
fast_inputs.Bit1:=FDI1;
fast_inputs.Bit2:=FDI2;

discrete_inputs.first_byte.Bit1:=DI1;
discrete_inputs.first_byte.Bit2:=DI2;
discrete_inputs.first_byte.Bit3:=DI3;
discrete_inputs.first_byte.Bit4:=DI4;
discrete_inputs.first_byte.Bit5:=DI5;
discrete_inputs.first_byte.Bit6:=DI6;
discrete_inputs.first_byte.Bit7:=DI7;
discrete_inputs.first_byte.Bit8:=DI8;
discrete_inputs.second_byte.Bit1:=DI9;
discrete_inputs.second_byte.Bit2:=DI10;
discrete_inputs.second_byte.Bit3:=DI11;
discrete_inputs.second_byte.Bit4:=DI12;
discrete_inputs.second_byte.Bit5:=DI13;
discrete_inputs.second_byte.Bit6:=DI14;
discrete_inputs.second_byte.Bit7:=DI15;
discrete_inputs.second_byte.Bit8:=DI16;

special_input.Bit1:=SI;

fast_outputs.Bit1:=FDO1;
fast_outputs.Bit2:=FDO2;
fast_outputs.Bit3:=FDO3;
fast_outputs.Bit4:=FDO4;

discrete_outputs.first_byte.Bit1:=DO1;
discrete_outputs.first_byte.Bit2:=DO2;
discrete_outputs.first_byte.Bit3:=DO3;
discrete_outputs.first_byte.Bit4:=DO4;
discrete_outputs.first_byte.Bit5:=DO5;
discrete_outputs.first_byte.Bit6:=DO6;
discrete_outputs.first_byte.Bit7:=DO7;
discrete_outputs.first_byte.Bit8:=DO8;

discrete_outputs.second_byte.Bit1:=DO9;
discrete_outputs.second_byte.Bit2:=DO10;
discrete_outputs.second_byte.Bit3:=DO11;
discrete_outputs.second_byte.Bit4:=DO12;
discrete_outputs.second_byte.Bit5:=DO13;
discrete_outputs.second_byte.Bit6:=DO14;
discrete_outputs.second_byte.Bit7:=DO15;
discrete_outputs.second_byte.Bit8:=DO16;

special_output.Bit1:=SO;
END_ACTION

(* POU PLC110_32/get_status_outputs, ST *)
FUNCTION_BLOCK get_status_outputs

VAR_INPUT
	fdo1:BOOL:=FALSE;
	fdo2:BOOL:=FALSE;
	fdo3:BOOL:=FALSE;
	fdo4:BOOL:=FALSE;
	do1:BOOL:=FALSE;
	do2:BOOL:=FALSE;
	do3:BOOL:=FALSE;
	do4:BOOL:=FALSE;
	do5:BOOL:=FALSE;
	do6:BOOL:=FALSE;
	do7:BOOL:=FALSE;
	do8:BOOL:=FALSE;
	do9:BOOL:=FALSE;
	do10:BOOL:=FALSE;
	do11:BOOL:=FALSE;
	do12:BOOL:=FALSE;
	do13:BOOL:=FALSE;
	do14:BOOL:=FALSE;
	do15:BOOL:=FALSE;
	do16:BOOL:=FALSE;
	sdo:BOOL:=FALSE;
END_VAR

VAR_OUTPUT
	get_status_outputs:classPLC32m2StatusOutputs;
END_VAR
get_status_outputs := get_status_outputs_def(fdo1, fdo2, fdo3, fdo4, do1, do2, do3, do4, do5, do6, do7, do8, do9, do10, do11, do12, do13, do14, do15, do16, sdo);
END_FUNCTION_BLOCK

(* POU PLC110_32/get_status_outputs_def, ST *)
FUNCTION get_status_outputs_def : classPLC32m2StatusOutputs

VAR_INPUT
	fdo1:BOOL:=FALSE;
	fdo2:BOOL:=FALSE;
	fdo3:BOOL:=FALSE;
	fdo4:BOOL:=FALSE;
	do1:BOOL:=FALSE;
	do2:BOOL:=FALSE;
	do3:BOOL:=FALSE;
	do4:BOOL:=FALSE;
	do5:BOOL:=FALSE;
	do6:BOOL:=FALSE;
	do7:BOOL:=FALSE;
	do8:BOOL:=FALSE;
	do9:BOOL:=FALSE;
	do10:BOOL:=FALSE;
	do11:BOOL:=FALSE;
	do12:BOOL:=FALSE;
	do13:BOOL:=FALSE;
	do14:BOOL:=FALSE;
	do15:BOOL:=FALSE;
	do16:BOOL:=FALSE;
	sdo:BOOL:=FALSE;
END_VAR
get_status_outputs_def.fast_outputs.Bit1:=fdo1;
get_status_outputs_def.fast_outputs.Bit2:=fdo2;
get_status_outputs_def.fast_outputs.Bit3:=fdo3;
get_status_outputs_def.fast_outputs.Bit4:=fdo4;

get_status_outputs_def.discrete_outputs.first_byte.Bit1:=do1;
get_status_outputs_def.discrete_outputs.first_byte.Bit2:=do2;
get_status_outputs_def.discrete_outputs.first_byte.Bit3:=do3;
get_status_outputs_def.discrete_outputs.first_byte.Bit4:=do4;
get_status_outputs_def.discrete_outputs.first_byte.Bit5:=do5;
get_status_outputs_def.discrete_outputs.first_byte.Bit6:=do6;
get_status_outputs_def.discrete_outputs.first_byte.Bit7:=do7;
get_status_outputs_def.discrete_outputs.first_byte.Bit8:=do8;
get_status_outputs_def.discrete_outputs.second_byte.Bit1:=do9;
get_status_outputs_def.discrete_outputs.second_byte.Bit2:=do10;
get_status_outputs_def.discrete_outputs.second_byte.Bit3:=do11;
get_status_outputs_def.discrete_outputs.second_byte.Bit4:=do12;
get_status_outputs_def.discrete_outputs.second_byte.Bit5:=do13;
get_status_outputs_def.discrete_outputs.second_byte.Bit6:=do14;
get_status_outputs_def.discrete_outputs.second_byte.Bit7:=do15;
get_status_outputs_def.discrete_outputs.second_byte.Bit8:=do16;

get_status_outputs_def.special_output.Bit1:=sdo;
END_FUNCTION

(* POU MB110_8.A/MB110_8a, ST *)
FUNCTION_BLOCK MB110_8a

VAR_INPUT
	ch1_error_code:WORD:=61447;
	ch1_value:REAL;
	ch2_error_code:WORD:=61447;
	ch2_value:REAL;
	ch3_error_code:WORD:=61447;
	ch3_value:REAL;
	ch4_error_code:WORD:=61447;
	ch4_value:REAL;
	ch5_error_code:WORD:=61447;
	ch5_value:REAL;
	ch6_error_code:WORD:=61447;
	ch6_value:REAL;
	ch7_error_code:WORD:=61447;
	ch7_value:REAL;
	ch8_error_code:WORD:=61447;
	ch8_value:REAL;
	settings:classSetAnalogInputsModule;
END_VAR

VAR_OUTPUT
	info:classInfoAnalogInputModule;
END_VAR
get_info_message;
END_FUNCTION_BLOCK
ACTION get_info_message:
info.channel1.error_message:=get_error_code(ch1_error_code);
info.channel2.error_message:=get_error_code(ch2_error_code);
info.channel3.error_message:=get_error_code(ch3_error_code);
info.channel4.error_message:=get_error_code(ch4_error_code);
info.channel5.error_message:=get_error_code(ch5_error_code);
info.channel6.error_message:=get_error_code(ch6_error_code);
info.channel7.error_message:=get_error_code(ch7_error_code);
info.channel8.error_message:=get_error_code(ch8_error_code);

info.channel1.current_value:=get_current_value(ch1_error_code,settings.ch1_set, ch1_value);
info.channel2.current_value:=get_current_value(ch2_error_code,settings.ch2_set, ch2_value);
info.channel3.current_value:=get_current_value(ch3_error_code,settings.ch3_set, ch3_value);
info.channel4.current_value:=get_current_value(ch4_error_code,settings.ch4_set, ch4_value);
info.channel5.current_value:=get_current_value(ch5_error_code,settings.ch5_set, ch5_value);
info.channel6.current_value:=get_current_value(ch6_error_code,settings.ch6_set, ch6_value);
info.channel7.current_value:=get_current_value(ch7_error_code,settings.ch7_set, ch7_value);
info.channel8.current_value:=get_current_value(ch8_error_code,settings.ch8_set, ch8_value);
END_ACTION

(* POU MB110_8.A/get_error_code, ST *)
FUNCTION get_error_code: STRING(79)
(* ï¿½ï¿½ï¿½ï¿½ï¿½ï¿½ï¿½ ï¿½ï¿½ï¿½ï¿½ï¿½ï¿½ï¿½ï¿½ï¿½ï¿½ï¿½ï¿½ï¿½ï¿½ ï¿½ï¿½ï¿½ï¿½ ï¿½ï¿½ï¿½ï¿½ï¿½ï¿½ ï¿½ï¿½ï¿½ï¿½ï¿½ï¿½ï¿½ï¿½ ï¿½ï¿½ï¿½ï¿½ï¿½ï¿½ï¿½ï¿½ï¿½ï¿½ï¿½ ï¿½ï¿½ï¿½ï¿½ï¿½ï¿½ ï¿½ï¿½ï¿½ï¿½ï¿½ï¿½ *)

VAR_INPUT
	code_error: WORD;
END_VAR

VAR
	error_message: STRING(79);
END_VAR
IF code_error=0
	THEN error_message := 'ï¿½ï¿½ï¿½ï¿½ï¿½ï¿½ï¿½ï¿½ï¿½ ï¿½ï¿½ï¿½ï¿½ï¿½ï¿½ï¿½';
ELSIF code_error = 61440
	THEN error_message := 'ï¿½ï¿½ï¿½ï¿½ï¿½ï¿½ï¿½ï¿½ ï¿½ï¿½ï¿½ï¿½ï¿½ï¿½ï¿½ï¿½ ï¿½ï¿½ï¿½ï¿½ï¿½ï¿½ï¿½';
ELSIF code_error = 61446
	THEN error_message := 'ï¿½ï¿½ï¿½ï¿½ï¿½ï¿½ ï¿½ï¿½ ï¿½ï¿½ï¿½ï¿½ï¿½ï¿½. ï¿½ï¿½ï¿½ï¿½ï¿½ ï¿½ï¿½ï¿½ï¿½ï¿½ï¿½ï¿½ï¿½ï¿½ï¿½ï¿½ ï¿½ï¿½ï¿½ï¿½ï¿½ï¿½ï¿½ ï¿½ï¿½ï¿½ï¿½ï¿½ï¿½ï¿½ï¿½ï¿½.';
ELSIF code_error = 61447
	THEN error_message := 'ï¿½ï¿½ï¿½ï¿½ï¿½ï¿½ ï¿½ï¿½ï¿½ï¿½ï¿½ï¿½ï¿½ï¿½.';
ELSIF code_error = 61448
	THEN error_message := 'ï¿½ï¿½ï¿½ï¿½ï¿½ï¿½ ï¿½ï¿½ï¿½ï¿½ï¿½ï¿½ï¿½ï¿½ï¿½ï¿½ï¿½ ï¿½ï¿½ï¿½ï¿½ï¿½ï¿½ï¿½ï¿½ï¿½ ï¿½ï¿½ï¿½ï¿½ï¿½ï¿½ ï¿½ï¿½.';
ELSIF code_error = 61449
	THEN error_message := 'ï¿½ï¿½ï¿½ï¿½ ï¿½ï¿½ï¿½ï¿½ï¿½ï¿½ï¿½ï¿½ï¿½ï¿½ï¿½ ï¿½ï¿½ï¿½ï¿½ï¿½ï¿½ï¿½ï¿½ï¿½ ï¿½ï¿½ï¿½ï¿½ï¿½ï¿½ ï¿½ï¿½.';
ELSIF code_error = 61450
	THEN error_message := 'ï¿½ï¿½ï¿½ï¿½ï¿½ï¿½ï¿½ï¿½ï¿½ï¿½ ï¿½ï¿½ï¿½ï¿½ï¿½ï¿½ï¿½ï¿½ ï¿½ï¿½ï¿½ï¿½ï¿½ï¿½ï¿½ ï¿½ï¿½ï¿½ï¿½ï¿½ï¿½.';
ELSIF code_error = 61451
	THEN error_message := 'ï¿½ï¿½ï¿½ï¿½ï¿½ï¿½ï¿½ï¿½ï¿½ï¿½ ï¿½ï¿½ï¿½ï¿½ï¿½ï¿½ï¿½ï¿½ ï¿½ï¿½ï¿½ï¿½ï¿½ï¿½ï¿½ ï¿½ï¿½ï¿½ï¿½.';
ELSIF code_error = 61452
	THEN error_message := 'ï¿½ï¿½ï¿½ï¿½ï¿½ï¿½ï¿½ï¿½ ï¿½ï¿½ï¿½ï¿½ï¿½ï¿½ï¿½ï¿½ï¿½ ï¿½ï¿½ï¿½ï¿½ï¿½ï¿½ï¿½.';
ELSIF code_error = 61453
	THEN error_message := 'ï¿½ï¿½ï¿½ï¿½ï¿½ ï¿½ï¿½ï¿½ï¿½ï¿½ï¿½ï¿½.';
ELSIF code_error = 61454
	THEN error_message := 'ï¿½ï¿½ï¿½ï¿½ï¿½ï¿½ï¿½ï¿½ï¿½ï¿½ ï¿½ï¿½ï¿½ï¿½ï¿½ ï¿½ ï¿½ï¿½ï¿½.';
ELSIF code_error = 61455
	THEN error_message := 'ï¿½ï¿½ï¿½ï¿½ï¿½ï¿½ï¿½ï¿½ï¿½ï¿½ï¿½ï¿½ ï¿½ï¿½ï¿½ï¿½ï¿½ï¿½ï¿½ï¿½ï¿½ï¿½ï¿½ï¿½ï¿½ ï¿½ï¿½ï¿½ï¿½ï¿½ï¿½ï¿½ï¿½ï¿½ï¿½ï¿½.';
ELSE
	error_message := 'Error not Found';
END_IF

get_error_code := error_message;
END_FUNCTION

(* POU MB110_8.A/get_current_value, ST *)
FUNCTION get_current_value : REAL
(* ï¿½ï¿½ï¿½ï¿½ï¿½ï¿½ï¿½ ï¿½ï¿½ï¿½ï¿½ï¿½ï¿½ï¿½ï¿½ï¿½ï¿½ï¿½ï¿½ï¿½ï¿½ï¿½ ï¿½ï¿½ï¿½ï¿½ï¿½ï¿½ ï¿½ ï¿½ï¿½ï¿½ ï¿½ ï¿½ï¿½ï¿½ï¿½ï¿½ï¿½ï¿½ï¿½ ï¿½ï¿½ï¿½ï¿½ *)

VAR_INPUT
	code_error:WORD;
	ch_set:classSetAnalogInputChannel;
	ch_value:REAL;
END_VAR
IF code_error = 0 THEN
	get_current_value := value_scaling(ch_value, get_set_Ain_value_params(ch_set));
ELSE
	(* ï¿½ï¿½ï¿½ï¿½ ï¿½ï¿½ï¿½ï¿½ï¿½ï¿½ ï¿½ï¿½ï¿½ï¿½ï¿½ï¿½ ï¿½ï¿½ï¿½ï¿½ï¿½ï¿½ ï¿½ï¿½ï¿½ï¿½ï¿½ï¿½ï¿½ ï¿½ï¿½ï¿½ï¿½ï¿½ï¿½ *)
	get_current_value := -8;
END_IF;
END_FUNCTION

(* POU function/value_scale/value_scaling, ST *)
FUNCTION value_scaling : REAL
(* ï¿½ï¿½ï¿½ï¿½ï¿½ï¿½ï¿½ ï¿½ï¿½ï¿½ï¿½ï¿½ï¿½ï¿½ï¿½ï¿½ï¿½ï¿½ï¿½ï¿½ï¿½ï¿½ ï¿½ï¿½ï¿½ï¿½ï¿½ *)

VAR_INPUT
	input_value: REAL;
	params_scales:classParamsValueScaling;
END_VAR

VAR
	A: REAL;
	B: REAL;
END_VAR
A := (params_scales.out_max - params_scales.out_min) / (params_scales.in_max - params_scales.in_min);
B := ((params_scales.out_min * params_scales.in_max) - (params_scales.out_max * params_scales.in_min)) / (params_scales.in_max - params_scales.in_min);

value_scaling := A * input_value + B;
END_FUNCTION

(* POU MB110_8.A/get_set_Ain_value_params, ST *)
FUNCTION get_set_Ain_value_params : classParamsValueScaling
(* ï¿½ï¿½ï¿½ï¿½ï¿½ï¿½ï¿½ï¿½ï¿½ï¿½ï¿½ï¿½ï¿½ï¿½ ï¿½ï¿½ ï¿½ï¿½ï¿½ï¿½ ï¿½ï¿½ï¿½ï¿½ï¿½ï¿½ï¿½ï¿½ ï¿½ï¿½ï¿½ï¿½ï¿½ ï¿½ ï¿½ï¿½ï¿½ï¿½ï¿½ï¿½ï¿½ï¿½ï¿½ ï¿½ï¿½ï¿½ï¿½ï¿½ï¿½ï¿½ï¿½ï¿½ï¿½ï¿½ï¿½ï¿½ï¿½ï¿½ *)

VAR_INPUT
	set:classSetAnalogInputChannel;
END_VAR
get_set_Ain_value_params.in_min:=set.ain_l;
get_set_Ain_value_params.in_max:=set.ain_h;
get_set_Ain_value_params.out_min:=set.analog_min_value;
get_set_Ain_value_params.out_max:=set.analog_max_value;
END_FUNCTION

(* POU MB110_8U/get_info_analog_outputs_module, ST *)
FUNCTION_BLOCK get_info_analog_outputs_module

VAR_INPUT
	ch1_current:REAL;
	ch2_current:REAL;
	ch3_current:REAL;
	ch4_current:REAL;
	ch5_current:REAL;
	ch6_current:REAL;
	ch7_current:REAL;
	ch8_current:REAL;
END_VAR

VAR_OUTPUT
	info:classAnalogOutputModule;
END_VAR
info.channel1.current_value := ch1_current;
info.channel2.current_value := ch2_current;
info.channel3.current_value := ch3_current;
info.channel4.current_value := ch4_current;
info.channel5.current_value := ch5_current;
info.channel6.current_value := ch6_current;
info.channel7.current_value := ch7_current;
info.channel8.current_value := ch8_current;
END_FUNCTION_BLOCK

(* POU MB110_8U/MY110_8u, ST *)
FUNCTION_BLOCK MY110_8u

VAR_INPUT
	info_current_channel:classAnalogOutputModule;
END_VAR

VAR_OUTPUT
	ch1_value:WORD;
	ch2_value:WORD;
	ch3_value:WORD;
	ch4_value:WORD;
	ch5_value:WORD;
	ch6_value:WORD;
	ch7_value:WORD;
	ch8_value:WORD;
END_VAR

VAR
	ch_ain_l: REAL := 4;  (* ï¿½ï¿½ï¿½ï¿½ï¿½ï¿½ï¿½ï¿½ ï¿½ï¿½ï¿½ï¿½ï¿½ï¿½ ï¿½ï¿½ï¿½ï¿½ï¿½ï¿½ï¿½ ï¿½ï¿½ï¿½ï¿½ï¿½ï¿½ï¿½ï¿½ ï¿½ï¿½ï¿½ï¿½ï¿½ï¿½ï¿½ï¿½ï¿½ *)
	ch_ain_h: REAL := 20;  (* ï¿½ï¿½ï¿½ï¿½ï¿½ï¿½ï¿½ï¿½ ï¿½ï¿½ï¿½ï¿½ï¿½ï¿½ï¿½ ï¿½ï¿½ï¿½ï¿½ï¿½ï¿½ï¿½ ï¿½ï¿½ï¿½ï¿½ï¿½ï¿½ï¿½ï¿½ ï¿½ï¿½ï¿½ï¿½ï¿½ï¿½ï¿½ï¿½ï¿½ *)
	ch_analog_min_value: REAL :=  0;  (* ï¿½ï¿½ï¿½ï¿½ï¿½ï¿½ ï¿½ï¿½ï¿½ï¿½ï¿½ï¿½ï¿½ ï¿½ï¿½ï¿½ *)
	ch_analog_max_value: REAL := 1000;  (* ï¿½ï¿½ï¿½ï¿½ï¿½ï¿½ï¿½ ï¿½ï¿½ï¿½ï¿½ï¿½ï¿½ï¿½ ï¿½ï¿½ï¿½ *)
	set_params:classParamsValueScaling;
END_VAR
set_params := get_params_value_scaling(ch_ain_l, ch_ain_h, ch_analog_min_value, ch_analog_max_value);

ch1_value := REAL_TO_INT(value_scaling(info_current_channel.channel1.current_value, set_params));
ch2_value := REAL_TO_INT(value_scaling(info_current_channel.channel2.current_value, set_params));
ch3_value := REAL_TO_INT(value_scaling(info_current_channel.channel3.current_value, set_params));
ch4_value := REAL_TO_INT(value_scaling(info_current_channel.channel4.current_value, set_params));
ch5_value := REAL_TO_INT(value_scaling(info_current_channel.channel5.current_value, set_params));
ch6_value := REAL_TO_INT(value_scaling(info_current_channel.channel6.current_value, set_params));
ch7_value := REAL_TO_INT(value_scaling(info_current_channel.channel7.current_value, set_params));
ch8_value := REAL_TO_INT(value_scaling(info_current_channel.channel8.current_value, set_params));
END_FUNCTION_BLOCK

(* POU function/value_scale/get_params_value_scaling, ST *)
FUNCTION get_params_value_scaling : classParamsValueScaling

VAR_INPUT
	in_min: REAL;
	in_max: REAL;
	out_min: REAL;
	out_max: REAL;
END_VAR
get_params_value_scaling.in_min := in_min;
get_params_value_scaling.in_max := in_max;
get_params_value_scaling.out_min := out_min;
get_params_value_scaling.out_max := out_max;
END_FUNCTION

(* POU MB110_8.A/SetChannelsAnalogInputsModule, ST *)
FUNCTION_BLOCK SetChannelsAnalogInputsModule

VAR_INPUT
	(* ï¿½ï¿½ï¿½ï¿½ï¿½ï¿½ï¿½ï¿½ï¿½ï¿½ï¿½ï¿½ï¿½ï¿½ï¿½ï¿½ ï¿½ï¿½ï¿½ï¿½ï¿½ï¿½ï¿½ï¿½ï¿½ ï¿½ï¿½ï¿½ï¿½ï¿½ï¿½ ï¿½ï¿½ï¿½ï¿½ï¿½ï¿½. ï¿½ï¿½. ï¿½ï¿½ï¿½ï¿½ï¿½ï¿½ï¿½ï¿½ï¿½ï¿½ ï¿½ï¿½ï¿½ï¿½ï¿½ï¿½ï¿½: ï¿½ï¿½ï¿½ï¿½ï¿½ï¿½ï¿½ï¿½ï¿½ï¿½. ï¿½ï¿½ï¿½ï¿½ï¿½ï¿½ï¿½ ï¿½.2 *)
	(* ï¿½ï¿½ï¿½ï¿½ï¿½ï¿½ï¿½ ï¿½ï¿½ï¿½ ï¿½ ï¿½ï¿½ï¿½ï¿½ï¿½ï¿½ï¿½ï¿½ ï¿½ï¿½ ï¿½ï¿½ï¿½ï¿½ï¿½ï¿½ï¿½ï¿½ï¿½: ï¿½ï¿½ï¿½ ï¿½ï¿½ï¿½ï¿½ï¿½ï¿½ï¿½ 4-20mA  *)

	ch1_ain_l: REAL := 0;  (* ï¿½ï¿½ï¿½ï¿½ï¿½ï¿½ï¿½ï¿½ Ain.L *)
	ch1_ain_h: REAL := 100;  (* ï¿½ï¿½ï¿½ï¿½ï¿½ï¿½ï¿½ï¿½ Ain.H *)
	ch1_analog_min_value: REAL := 4;  (* ï¿½ï¿½ï¿½ï¿½ï¿½ï¿½ï¿½ï¿½ ï¿½ï¿½ï¿½ï¿½ï¿½ï¿½ ï¿½ï¿½ï¿½ï¿½ï¿½ï¿½ï¿½ ï¿½ï¿½ï¿½ï¿½ï¿½ï¿½ï¿½ *)
	ch1_analog_max_value: REAL := 20;  (* ï¿½ï¿½ï¿½ï¿½ï¿½ï¿½ï¿½ï¿½ ï¿½ï¿½ï¿½ï¿½ï¿½ï¿½ï¿½ ï¿½ï¿½ï¿½ï¿½ï¿½ï¿½ï¿½ ï¿½ï¿½ï¿½ï¿½ï¿½ï¿½ï¿½ *)

	ch2_ain_l: REAL := 0;  (* ï¿½ï¿½ï¿½ï¿½ï¿½ï¿½ï¿½ï¿½ Ain.L *)
	ch2_ain_h: REAL := 100;  (* ï¿½ï¿½ï¿½ï¿½ï¿½ï¿½ï¿½ï¿½ Ain.H *)
	ch2_analog_min_value: REAL := 4;  (* ï¿½ï¿½ï¿½ï¿½ï¿½ï¿½ï¿½ï¿½ ï¿½ï¿½ï¿½ï¿½ï¿½ï¿½ ï¿½ï¿½ï¿½ï¿½ï¿½ï¿½ï¿½ ï¿½ï¿½ï¿½ï¿½ï¿½ï¿½ï¿½ *)
	ch2_analog_max_value: REAL := 20;  (* ï¿½ï¿½ï¿½ï¿½ï¿½ï¿½ï¿½ï¿½ ï¿½ï¿½ï¿½ï¿½ï¿½ï¿½ï¿½ ï¿½ï¿½ï¿½ï¿½ï¿½ï¿½ï¿½ ï¿½ï¿½ï¿½ï¿½ï¿½ï¿½ï¿½ *)

	ch3_ain_l: REAL := 0;  (* ï¿½ï¿½ï¿½ï¿½ï¿½ï¿½ï¿½ï¿½ Ain.L *)
	ch3_ain_h: REAL := 100;  (* ï¿½ï¿½ï¿½ï¿½ï¿½ï¿½ï¿½ï¿½ Ain.H *)
	ch3_analog_min_value: REAL := 4;  (* ï¿½ï¿½ï¿½ï¿½ï¿½ï¿½ï¿½ï¿½ ï¿½ï¿½ï¿½ï¿½ï¿½ï¿½ ï¿½ï¿½ï¿½ï¿½ï¿½ï¿½ï¿½ ï¿½ï¿½ï¿½ï¿½ï¿½ï¿½ï¿½ *)
	ch3_analog_max_value: REAL := 20;  (* ï¿½ï¿½ï¿½ï¿½ï¿½ï¿½ï¿½ï¿½ ï¿½ï¿½ï¿½ï¿½ï¿½ï¿½ï¿½ ï¿½ï¿½ï¿½ï¿½ï¿½ï¿½ï¿½ ï¿½ï¿½ï¿½ï¿½ï¿½ï¿½ï¿½ *)

	ch4_ain_l: REAL := 0;  (* ï¿½ï¿½ï¿½ï¿½ï¿½ï¿½ï¿½ï¿½ Ain.L *)
	ch4_ain_h: REAL := 100;  (* ï¿½ï¿½ï¿½ï¿½ï¿½ï¿½ï¿½ï¿½ Ain.H *)
	ch4_analog_min_value: REAL := 4;  (* ï¿½ï¿½ï¿½ï¿½ï¿½ï¿½ï¿½ï¿½ ï¿½ï¿½ï¿½ï¿½ï¿½ï¿½ ï¿½ï¿½ï¿½ï¿½ï¿½ï¿½ï¿½ ï¿½ï¿½ï¿½ï¿½ï¿½ï¿½ï¿½ *)
	ch4_analog_max_value: REAL := 20;  (* ï¿½ï¿½ï¿½ï¿½ï¿½ï¿½ï¿½ï¿½ ï¿½ï¿½ï¿½ï¿½ï¿½ï¿½ï¿½ ï¿½ï¿½ï¿½ï¿½ï¿½ï¿½ï¿½ ï¿½ï¿½ï¿½ï¿½ï¿½ï¿½ï¿½ *)

	ch5_ain_l: REAL := 0;  (* ï¿½ï¿½ï¿½ï¿½ï¿½ï¿½ï¿½ï¿½ Ain.L *)
	ch5_ain_h: REAL := 100;  (* ï¿½ï¿½ï¿½ï¿½ï¿½ï¿½ï¿½ï¿½ Ain.H *)
	ch5_analog_min_value: REAL := 4;  (* ï¿½ï¿½ï¿½ï¿½ï¿½ï¿½ï¿½ï¿½ ï¿½ï¿½ï¿½ï¿½ï¿½ï¿½ ï¿½ï¿½ï¿½ï¿½ï¿½ï¿½ï¿½ ï¿½ï¿½ï¿½ï¿½ï¿½ï¿½ï¿½ *)
	ch5_analog_max_value: REAL := 20;  (* ï¿½ï¿½ï¿½ï¿½ï¿½ï¿½ï¿½ï¿½ ï¿½ï¿½ï¿½ï¿½ï¿½ï¿½ï¿½ ï¿½ï¿½ï¿½ï¿½ï¿½ï¿½ï¿½ ï¿½ï¿½ï¿½ï¿½ï¿½ï¿½ï¿½ *)

	ch6_ain_l: REAL := 0;  (* ï¿½ï¿½ï¿½ï¿½ï¿½ï¿½ï¿½ï¿½ Ain.L *)
	ch6_ain_h: REAL := 100;  (* ï¿½ï¿½ï¿½ï¿½ï¿½ï¿½ï¿½ï¿½ Ain.H *)
	ch6_analog_min_value: REAL := 4;  (* ï¿½ï¿½ï¿½ï¿½ï¿½ï¿½ï¿½ï¿½ ï¿½ï¿½ï¿½ï¿½ï¿½ï¿½ ï¿½ï¿½ï¿½ï¿½ï¿½ï¿½ï¿½ ï¿½ï¿½ï¿½ï¿½ï¿½ï¿½ï¿½ *)
	ch6_analog_max_value: REAL := 20;  (* ï¿½ï¿½ï¿½ï¿½ï¿½ï¿½ï¿½ï¿½ ï¿½ï¿½ï¿½ï¿½ï¿½ï¿½ï¿½ ï¿½ï¿½ï¿½ï¿½ï¿½ï¿½ï¿½ ï¿½ï¿½ï¿½ï¿½ï¿½ï¿½ï¿½ *)

	ch7_ain_l: REAL := 0;  (* ï¿½ï¿½ï¿½ï¿½ï¿½ï¿½ï¿½ï¿½ Ain.L *)
	ch7_ain_h: REAL := 100;  (* ï¿½ï¿½ï¿½ï¿½ï¿½ï¿½ï¿½ï¿½ Ain.H *)
	ch7_analog_min_value: REAL := 4;  (* ï¿½ï¿½ï¿½ï¿½ï¿½ï¿½ï¿½ï¿½ ï¿½ï¿½ï¿½ï¿½ï¿½ï¿½ ï¿½ï¿½ï¿½ï¿½ï¿½ï¿½ï¿½ ï¿½ï¿½ï¿½ï¿½ï¿½ï¿½ï¿½ *)
	ch7_analog_max_value: REAL := 20;  (* ï¿½ï¿½ï¿½ï¿½ï¿½ï¿½ï¿½ï¿½ ï¿½ï¿½ï¿½ï¿½ï¿½ï¿½ï¿½ ï¿½ï¿½ï¿½ï¿½ï¿½ï¿½ï¿½ ï¿½ï¿½ï¿½ï¿½ï¿½ï¿½ï¿½ *)

	ch8_ain_l: REAL := 0;  (* ï¿½ï¿½ï¿½ï¿½ï¿½ï¿½ï¿½ï¿½ Ain.L *)
	ch8_ain_h: REAL := 100;  (* ï¿½ï¿½ï¿½ï¿½ï¿½ï¿½ï¿½ï¿½ Ain.H *)
	ch8_analog_min_value: REAL := 4;  (* ï¿½ï¿½ï¿½ï¿½ï¿½ï¿½ï¿½ï¿½ ï¿½ï¿½ï¿½ï¿½ï¿½ï¿½ ï¿½ï¿½ï¿½ï¿½ï¿½ï¿½ï¿½ ï¿½ï¿½ï¿½ï¿½ï¿½ï¿½ï¿½ *)
	ch8_analog_max_value: REAL := 20;  (* ï¿½ï¿½ï¿½ï¿½ï¿½ï¿½ï¿½ï¿½ ï¿½ï¿½ï¿½ï¿½ï¿½ï¿½ï¿½ ï¿½ï¿½ï¿½ï¿½ï¿½ï¿½ï¿½ ï¿½ï¿½ï¿½ï¿½ï¿½ï¿½ï¿½ *)
END_VAR

VAR_OUTPUT
	settings:classSetAnalogInputsModule;
END_VAR
get_settings;
END_FUNCTION_BLOCK
ACTION get_settings:
settings.ch1_set := get_setAin(ch1_ain_l, ch1_ain_h, ch1_analog_min_value, ch1_analog_max_value);
settings.ch2_set := get_setAin(ch2_ain_l, ch2_ain_h, ch2_analog_min_value, ch2_analog_max_value);
settings.ch3_set := get_setAin(ch3_ain_l, ch3_ain_h, ch3_analog_min_value, ch3_analog_max_value);
settings.ch4_set := get_setAin(ch4_ain_l, ch4_ain_h, ch4_analog_min_value, ch4_analog_max_value);
settings.ch5_set := get_setAin(ch5_ain_l, ch5_ain_h, ch5_analog_min_value, ch5_analog_max_value);
settings.ch6_set := get_setAin(ch6_ain_l, ch6_ain_h, ch6_analog_min_value, ch6_analog_max_value);
settings.ch7_set := get_setAin(ch7_ain_l, ch7_ain_h, ch7_analog_min_value, ch7_analog_max_value);
settings.ch8_set := get_setAin(ch8_ain_l, ch8_ain_h, ch8_analog_min_value, ch8_analog_max_value);
END_ACTION

(* POU MB110_8.A/get_setAin, ST *)
FUNCTION get_setAin : classSetAnalogInputChannel
(* ï¿½ï¿½ï¿½ï¿½ï¿½ï¿½ï¿½ï¿½ï¿½ ï¿½ï¿½ï¿½ï¿½ï¿½ï¿½ï¿½ï¿½ ï¿½ dataclass *)

VAR_INPUT
	ch_ain_l: REAL := 0;  (* ï¿½ï¿½ï¿½ï¿½ï¿½ï¿½ï¿½ï¿½ Ain.L *)
	ch_ain_h: REAL := 100;  (* ï¿½ï¿½ï¿½ï¿½ï¿½ï¿½ï¿½ï¿½ Ain.H *)
	ch_analog_min_value: REAL := 4;  (* ï¿½ï¿½ï¿½ï¿½ï¿½ï¿½ï¿½ï¿½ ï¿½ï¿½ï¿½ï¿½ï¿½ï¿½ ï¿½ï¿½ï¿½ï¿½ï¿½ï¿½ï¿½ ï¿½ï¿½ï¿½ï¿½ï¿½ï¿½ï¿½ *)
	ch_analog_max_value: REAL := 20;  (* ï¿½ï¿½ï¿½ï¿½ï¿½ï¿½ï¿½ï¿½ ï¿½ï¿½ï¿½ï¿½ï¿½ï¿½ï¿½ ï¿½ï¿½ï¿½ï¿½ï¿½ï¿½ï¿½ ï¿½ï¿½ï¿½ï¿½ï¿½ï¿½ï¿½ *)
END_VAR
get_setAin.ain_l:=ch_ain_l;
get_setAin.ain_h:=ch_ain_h;
get_setAin.analog_min_value:=ch_analog_min_value;
get_setAin.analog_max_value:=ch_analog_max_value;
END_FUNCTION

(* POU PressureSensor_4_20ma/CurrentSensorPressure_4_20, ST *)
FUNCTION_BLOCK CurrentSensorPressure_4_20

VAR_INPUT
	current_value:REAL;  (*ï¿½ï¿½ï¿½ï¿½ï¿½ï¿½ï¿½ï¿½ ï¿½ï¿½ï¿½ï¿½ 4-20ï¿½ï¿½ *)
	set:classSetPressureSensor4_20;  (* ï¿½ï¿½ï¿½ï¿½ï¿½ï¿½ï¿½ ï¿½ ï¿½ï¿½ï¿½ï¿½ï¿½ï¿½ ï¿½ï¿½ï¿½ï¿½ï¿½ï¿½ï¿½ ï¿½ï¿½ï¿½ï¿½ï¿½ï¿½ï¿½ï¿½ *)
END_VAR

VAR_OUTPUT
	pressure:REAL;  (* ï¿½ï¿½ï¿½ï¿½ï¿½ï¿½ï¿½ï¿½ ï¿½ï¿½ ï¿½ï¿½ï¿½ï¿½ï¿½ï¿½ *)
END_VAR
pressure:=value_scaling(current_value, get_set_sensor_value_params(set));
END_FUNCTION_BLOCK

(* POU PressureSensor_4_20ma/get_set_sensor_value_params, ST *)
FUNCTION get_set_sensor_value_params : classParamsValueScaling

VAR_INPUT
	sensor_set:classSetPressureSensor4_20;
END_VAR
get_set_sensor_value_params.in_min := sensor_set.min_current_range;
get_set_sensor_value_params.in_max := sensor_set.max_current_range;
get_set_sensor_value_params.out_min := sensor_set.min_measure_range;
get_set_sensor_value_params.out_max := sensor_set.max_measure_range;
END_FUNCTION

(* POU Invertor_Drive/InvertorDrive, ST *)
FUNCTION_BLOCK InvertorDrive
(* Function block implementation invertor drive. *)

VAR_INPUT
(* discrete inputs *)
	start: BOOL := FALSE;
	reset_fault: BOOL := FALSE;
	low_pressure_in: BOOL;  (* external alarm *)
	high_pressure_out: BOOL;  (* external alrm *)
(* discrete outputs *)
	status_run: BOOL;
	status_alarm: BOOL;
(* analog inputs *)
	ain_value: REAL := 0;  (* mA or V *)
(* analog outputs *)
	aout_value: REAL := 0;
(* PID settings *)
	auto: BOOL := FALSE;
	direct_logic: BOOL := TRUE;  (* flag forward/reverse control, reverse control: if input value less set point, output value to less. forward control: if input value less set point, output value to more. *)
	set_point: REAL := 0;  (* set point, measure system in input value control. *)
	P: REAL := 2;  (* proporcional value of PID, if more, out value fasted. *)
	I: INT := 10;  (* integral value of PID, seconds *)
	D:INT := 0;  (* differential value PID, seconds *)

(* limit work frequency *)
	manual: REAL := 0; (* set output value in manual mode, Hz*)
	min_range: REAL := 15;  (* min value in manual mode, Hz*)
	max_range: REAL := 50;  (* max value in manual mode, Hz*)

(* status invertor in work *)
	active: BOOL := FALSE;  (* statis active invertor drive. *)
	system_alarm: BOOL; (* alarm manager alarm_on *)
END_VAR

VAR_OUTPUT
	info: classInfoInvertorDrive;
	settings_pid: classSetPid;
END_VAR

VAR
	invertor_drive: classInvertorDrive;
    set_auto: classSetAutoInvertorDrive;
	set_frequency: classSetLimitFrequency;
	set_pid: classSetPid;

	discrete_inputs: classInvertorDriveDiscreteInputs;
	discrete_outputs: classInvertorDriveDiscreteOutputs;
	analog_inputs: classInvertorDriveAnalogInputs;
	analog_outputs: classInvertorDriveAnalogOutputs;

	overflow: BOOL := FALSE; (* overflow integral value of PID *)

	external_alarm:STRING(79); (* message of external alarm. *)

	info_alarm: classAlarmInvertorDrive;
END_VAR
init;

info_alarm.external_alarm := get_external_alarm(
	discrete_inputs.low_pressure_in, discrete_inputs.high_pressure_out
);

get_PID_set;

get_infomessage;
END_FUNCTION_BLOCK
ACTION get_infoMessage:
info.active := active;
info.set_pid := set_pid;
info.alarm.external_alarm := info_alarm.external_alarm;

IF discrete_outputs.status_alarm THEN
	info_alarm.fault_invertor_drive := 'Alarm invertor drive!';
	analog_outputs.out_frequency := 0;
ELSE
	info_alarm.fault_invertor_drive := 'No alarm';
END_IF;

info.alarm.fault_invertor_drive := info_alarm.fault_invertor_drive;

IF discrete_outputs.status_run THEN
	info.status_run := 'Run';

ELSE
	info.status_run := 'Stopped';
	analog_outputs.out_frequency := 0;
END_IF;

(* converted frequency in current value of 4-20 mA *)
info.frequency := analog_outputs.out_frequency;
info.aout_frequency := value_scaling(analog_outputs.out_frequency, get_params_value_scaling(0, 50, 4, 20));

IF info.alarm.external_alarm  <> 'GOOD' THEN
	discrete_inputs.start := FALSE;
ELSIF info.alarm.fault_invertor_drive <> 'No alarm' THEN
	discrete_inputs.start := FALSE;
ELSIF system_alarm <> 0 THEN
	discrete_inputs.start := FALSE;
ELSE
	discrete_inputs.start := invertor_drive.discrete_inputs.start;
END_IF;

info.reset_fault := discrete_inputs.reset_fault;

info.run := discrete_inputs.start;
END_ACTION
ACTION get_PID_set:
analog_inputs := invertor_drive.analog_input;
set_auto := invertor_drive.set.set_auto;
set_frequency := invertor_drive.set.set_frequency;

overflow := FALSE; (* this place for realise reset integral value of PID *) 

set_pid := get_set_pid(
	set_auto.direct_logic,
	set_auto.value,
	set_auto.set_point,
	set_auto.P,
	set_auto.I,
	set_auto.D,
	set_frequency.manual,
	0,
	set_frequency.min_range,
	set_frequency.max_range,
	NOT set_auto.auto,
	overflow
);

settings_pid := set_pid;
END_ACTION
ACTION init:
invertor_drive.analog_input.set_frequency := ain_value;
invertor_drive.analog_output.out_frequency := aout_value;

invertor_drive.discrete_inputs.start := start;
invertor_drive.discrete_inputs.reset_fault := reset_fault;
invertor_drive.discrete_inputs.low_pressure_in := low_pressure_in;
invertor_drive.discrete_inputs.high_pressure_out := high_pressure_out;

invertor_drive.discrete_outputs.status_run := status_run;
invertor_drive.discrete_outputs.status_alarm := status_alarm;

invertor_drive.set.set_frequency.min_range := min_range;
invertor_drive.set.set_frequency.max_range := max_range;

invertor_drive.set.set_auto.auto := auto;
invertor_drive.set.set_auto.direct_logic := direct_logic;
invertor_drive.set.set_auto.set_point := set_point;
invertor_drive.set.set_auto.value := ain_value;
invertor_drive.set.set_auto.P := P;
invertor_drive.set.set_auto.I := I;
invertor_drive.set.set_auto.D := D;

invertor_drive.set.set_frequency.manual := manual;
invertor_drive.set.set_frequency.min_range := min_range;
invertor_drive.set.set_frequency.max_range := max_range;

discrete_inputs := invertor_drive.discrete_inputs;
discrete_outputs := invertor_drive.discrete_outputs;
analog_outputs := invertor_drive.analog_output;
END_ACTION

(* POU Invertor_Drive/get_external_alarm, ST *)
FUNCTION get_external_alarm : STRING(79)
(* ï¿½ï¿½ï¿½ï¿½ï¿½ï¿½ï¿½ï¿½ï¿½ ï¿½ï¿½ï¿½ï¿½ï¿½ï¿½ï¿½ï¿½ï¿½ ï¿½ï¿½ï¿½ï¿½ï¿½ï¿½ ï¿½ï¿½ ï¿½ï¿½ï¿½ï¿½ï¿½ï¿½ ï¿½ï¿½ï¿½ï¿½ ï¿½ï¿½ï¿½ ï¿½ï¿½ï¿½ï¿½ï¿½ï¿½ï¿½ï¿½ï¿½ï¿½ ï¿½ï¿½ï¿½ï¿½ï¿½ï¿½ï¿½ï¿½ *)
VAR_INPUT
	low_pressure_in:BOOL;
	high_pressure_out:BOOL;
END_VAR
IF low_pressure_in THEN
	get_external_alarm:='ï¿½ï¿½ï¿½ï¿½ï¿½ï¿½ ï¿½ï¿½ï¿½ï¿½ï¿½ï¿½ï¿½ï¿½ ï¿½ï¿½ ï¿½ï¿½ï¿½ï¿½ï¿½';
ELSIF high_pressure_out THEN
	get_external_alarm:='ï¿½ï¿½ï¿½ï¿½ï¿½ï¿½ï¿½ ï¿½ï¿½ï¿½ï¿½ï¿½ï¿½ï¿½ï¿½ ï¿½ï¿½ ï¿½ï¿½ï¿½ï¿½ï¿½ï¿½';
ELSE
	get_external_alarm:='GOOD';
END_IF;
END_FUNCTION

(* POU PID_regulator/get_set_pid, ST *)
FUNCTION get_set_pid : classSetPid

VAR_INPUT
	direct_logic:BOOL:=TRUE;
	actual:REAL;
	set_point:REAL;
	P:REAL:=2;  (* ï¿½ï¿½ï¿½ï¿½ï¿½ï¿½ï¿½ï¿½ï¿½ï¿½ï¿½ï¿½ï¿½ï¿½ï¿½ï¿½ ï¿½ï¿½ï¿½ï¿½ï¿½ï¿½ï¿½ï¿½ï¿½ï¿½ï¿½ ï¿½ï¿½ï¿½ï¿½ï¿½ï¿½ï¿½ï¿½ï¿½ï¿½, ï¿½ï¿½ï¿½ ï¿½ï¿½ï¿½ï¿½ï¿½ï¿½ï¿½ï¿½ï¿½ï¿½ ï¿½ï¿½ï¿½ï¿½ï¿½ ï¿½ï¿½ï¿½ï¿½ï¿½ï¿½ï¿½ï¿½ï¿½ï¿½ ï¿½ï¿½ï¿½ï¿½ï¿½ï¿½ï¿½ï¿½ï¿½ï¿½ ï¿½ï¿½ï¿½ï¿½ï¿½ï¿½ï¿½*)
	I:INT:=10;  (* ï¿½ï¿½ï¿½ï¿½ï¿½ï¿½ï¿½ï¿½ï¿½ï¿½ï¿½ï¿½ ï¿½ï¿½ï¿½ï¿½ï¿½ï¿½ï¿½ï¿½ï¿½ï¿½ï¿½ ï¿½ï¿½ï¿½ï¿½ï¿½ï¿½ï¿½ï¿½ï¿½ï¿½, ï¿½ï¿½ï¿½ï¿½ï¿½ ï¿½ ï¿½ï¿½ï¿½ï¿½ï¿½ï¿½ï¿½ï¿½ *)
	D:INT:=0;  (* ï¿½ï¿½ï¿½ï¿½ï¿½ï¿½ï¿½ï¿½ï¿½ï¿½ï¿½ï¿½ï¿½ï¿½ï¿½ï¿½ ï¿½ï¿½ï¿½ï¿½ï¿½ï¿½ï¿½ï¿½ï¿½ï¿½ï¿½ ï¿½ï¿½ï¿½ï¿½ï¿½ï¿½ï¿½ï¿½ï¿½ï¿½, ï¿½ï¿½ï¿½ï¿½ï¿½ ï¿½ ï¿½ï¿½ï¿½ï¿½ï¿½ï¿½ï¿½ï¿½ *)
	Y_manual:REAL:=0;  (* Hz *)
	Y_offset:REAL:=0;
	Y_min:REAL;
	Y_max:REAL;
	manual:BOOL:=TRUE;  (* ï¿½ï¿½ï¿½ï¿½ï¿½ï¿½ï¿½ï¿½ï¿½ï¿½ï¿½ ï¿½ï¿½ï¿½ï¿½ï¿½ï¿½ï¿½ï¿½ ï¿½ï¿½ï¿½ï¿½ï¿½ï¿½ ï¿½ï¿½ï¿½ï¿½ï¿½ *)
	reset:BOOL:=FALSE;
END_VAR
IF direct_logic = TRUE THEN
	get_set_pid.actual := actual;
	get_set_pid.set_point := set_point;
ELSE
	get_set_pid.actual := set_point;
	get_set_pid.set_point := actual;
END_IF;

get_set_pid.P := P;
get_set_pid.I := I;
get_set_pid.D := D;
get_set_pid.Y_manual := Y_manual;
get_set_pid.Y_offset := Y_offset;
get_set_pid.Y_min := Y_min;
get_set_pid.Y_max := Y_max;
get_set_pid.manual := manual;
get_set_pid.reset := reset;
END_FUNCTION

(* POU PID_regulator/params_in_set_PID, ST *)
FUNCTION_BLOCK params_in_set_PID

VAR_INPUT
	set:classSetPid;
END_VAR

VAR_OUTPUT
	actual:REAL;
	set_point:REAL;
	P:REAL;
	I:REAL;
	D:REAL;
	Y_manual:REAL;
	Y_offset:REAL;
	Y_min:REAL;
	Y_max:REAL;
	manual:BOOL;
	reset:BOOL;
END_VAR
actual := set.actual;
set_point := set.set_point;
P := set.P;
I := set.I;
D := set.D;
Y_manual := set.Y_manual;
Y_offset := set.Y_offset;
Y_min := set.Y_min;
Y_max := set.Y_max;
manual := set.manual;
reset := set.reset;
END_FUNCTION_BLOCK

(* POU single_mode/Single, ST *)
FUNCTION_BLOCK Single
(* Function block implementation single mode. *)

VAR_INPUT
    enable: BOOL; (* Enable single mode *)
    pivot_pump: INT; (* pivot pump *)
    info_invertor_drive1: classInfoInvertorDrive;
    info_invertor_drive2: classInfoInvertorDrive;
    info_invertor_drive3: classInfoInvertorDrive;
    info_invertor_drive4: classInfoInvertorDrive;
    info_invertor_drive5: classInfoInvertorDrive;
    info_invertor_drive6: classInfoInvertorDrive;
    info_invertor_drive7: classInfoInvertorDrive;
    info_invertor_drive8: classInfoInvertorDrive;
END_VAR

VAR_OUTPUT
    info_single: classInfoSingle; (* info mode *)
END_VAR

VAR
    pivot: INT;
    pumps: ARRAY[1..8] OF BOOL;
END_VAR
pumps[1] := get_active(info_invertor_drive1);
pumps[2] := get_active(info_invertor_drive2);
pumps[3] := get_active(info_invertor_drive3);
pumps[4] := get_active(info_invertor_drive4);
pumps[5] := get_active(info_invertor_drive5);
pumps[6] := get_active(info_invertor_drive6);
pumps[7] := get_active(info_invertor_drive7);
pumps[8] := get_active(info_invertor_drive8);

pivot := pivot_pump;
IF pivot = 0 THEN
	enable := FALSE;
    info_single.error_code:=8;
END_IF;

IF enable THEN
    IF pumps[pivot] THEN
        info_single.pivot_pump := pivot;
        info_single.start_pump := pumps[pivot];
        info_single.error_code := 0;
        info_single.message := 'Select pump in work'; (* Выбранный насос в работе. *)
    ELSE
        info_single.pivot_pump := -8;
        info_single.start_pump := FALSE;
        info_single.error_code := 6;
        info_single.message := 'Select pump is not active!'; (* Выбранный насос не активен! *)
    END_IF;
      
ELSE
    info_single.pivot_pump := -8;
    info_single.start_pump := FALSE;
    info_single.error_code := 0; (* bug *)
    info_single.message := 'Single mode is not activate'; (* Режим работы одного насоса не активен. *)
END_IF;
END_FUNCTION_BLOCK

(* POU Invertor_Drive/get_active, ST *)
FUNCTION get_active : BOOL

VAR_INPUT
	info_invertor_drive:classInfoInvertorDrive;
END_VAR
get_active:=info_invertor_drive.active;
END_FUNCTION

(* POU cycle_mode/cycle, ST *)
FUNCTION_BLOCK cycle
(* Function block implementation cycle mode. *)

VAR_INPUT
	enable:BOOL;
	set_timer:TIME;
	info_invertor_drive1: classInfoInvertorDrive;
    info_invertor_drive2: classInfoInvertorDrive;
    info_invertor_drive3: classInfoInvertorDrive;
    info_invertor_drive4: classInfoInvertorDrive;
    info_invertor_drive5: classInfoInvertorDrive;
    info_invertor_drive6: classInfoInvertorDrive;
    info_invertor_drive7: classInfoInvertorDrive;
    info_invertor_drive8: classInfoInvertorDrive;
	END_VAR

VAR_OUTPUT
	info_cycle:classInfoCycle;
END_VAR
VAR
	pumps: ARRAY [1..8] OF BOOL;
	i: INT := 8;
	start_timer: TIME:=t#0ms;
	start_delay:TON;
	in: BOOL;

	working_time:TIME;
	Q:BOOL;
	n: INT;
END_VAR
pumps[1] := get_active(info_invertor_drive1);
pumps[2] := get_active(info_invertor_drive2);
pumps[3] := get_active(info_invertor_drive3);
pumps[4] := get_active(info_invertor_drive4);
pumps[5] := get_active(info_invertor_drive5);
pumps[6] := get_active(info_invertor_drive6);
pumps[7] := get_active(info_invertor_drive7);
pumps[8] := get_active(info_invertor_drive8);

n:=i;

IF pumps[i] = FALSE THEN
	i := i + 1;
END_IF;

IF  start_timer = t#0ms THEN
	start_timer := get_systime();
	in := TRUE;
END_IF;

working_time := work_time(start_timer);


IF working_time >= set_timer THEN
	in := FALSE;
	i := i + 1;
	start_timer := t#0ms;
END_IF;

start_delay(IN:=in, PT:=t#3s);
Q := start_delay.Q;

IF i > 8 THEN
	i := 1;
END_IF;

IF enable THEN
	info_cycle.working_time := working_time;
	info_cycle.run_timer := Q;
	info_cycle.pump_number := n;
ELSE
	info_cycle.working_time := T#0s;
	info_cycle.run_timer := FALSE;
	info_cycle.pump_number := 1;
	start_timer := t#0s;
END_IF;
info_cycle.error_code := 0;
END_FUNCTION_BLOCK

(* POU cycle_mode/get_systime, ST *)
FUNCTION get_systime : TIME

VAR_INPUT
END_VAR
get_systime:=TIME();
END_FUNCTION

(* POU cycle_mode/work_time, ST *)
FUNCTION work_time : TIME

VAR_INPUT
	start:TIME;
END_VAR
work_time:=TIME() - start;
END_FUNCTION

(* POU cascade_mode/cascade, ST *)
FUNCTION_BLOCK cascade
(* Functional block implementation cascade mode. *)
VAR_INPUT
	enable:BOOL;
	set_pressure:REAL;
	in_pressure: REAL;
	pivot_pump: INT;
	delay_on:TIME := t#30s;
	delay_off:TIME := t#30s;
    
	info_invertor_drive1: classInfoInvertorDrive;
    info_invertor_drive2: classInfoInvertorDrive;
    info_invertor_drive3: classInfoInvertorDrive;
    info_invertor_drive4: classInfoInvertorDrive;
    info_invertor_drive5: classInfoInvertorDrive;
    info_invertor_drive6: classInfoInvertorDrive;
    info_invertor_drive7: classInfoInvertorDrive;
    info_invertor_drive8: classInfoInvertorDrive;
END_VAR

VAR_OUTPUT
	info_cascade:classInfoCascade;
END_VAR

VAR
	pumps: ARRAY [1..8] OF BOOL;
	cascade_pumps: ARRAY [1..8] OF classInfoCascadePump;
	pivot: INT;
	i: INT:=1;
	error_message: STRING(79):= 'NOT GOOD';
	start_time: TIME:=t#0s;
	work_time: TIME;
	len_pumps: INT;
	index_active_pumps:ARRAY [1..8] OF INT;
	len_active_pumps: INT;
	index_pivot: INT;
	histeresys: REAL := 0.2 (* histeresys set pressure *);
	error_code:WORD;
END_VAR
pivot := pivot_pump;

IF pivot = 0 THEN
	check_pivot;
ELSE
    check_active_pumps;
END_IF;

IF len_active_pumps > 1  AND index_pivot <> 0 THEN
    cascade_on;
ELSIF len_active_pumps = 1 AND index_pivot <> 0 THEN
    i := index_pivot;
	error_code := 4;
    error_message := 'cascade mode excpected more one active pumps, but got less';
ELSIF index_pivot = 0 THEN
	error_code := 5;
	error_message := 'pivot pump not active';
END_IF;

get_info_message;
END_FUNCTION_BLOCK
ACTION cascade_on:
error_code := 0;
error_message := 'GOOD';

(* inspect bounds array. *)

IF i = 1 AND i = index_pivot THEN
	i := pivot + 1;
ELSIF i = len_active_pumps AND  i = index_pivot THEN
	i := len_active_pumps - 1;
END_IF;

(* start pivot pump. *)
IF INT_TO_BOOL(index_pivot) THEN
	cascade_pumps[pivot].cascade_pump := TRUE;
END_IF;

IF start_time = t#0s THEN
	start_time := TIME();
END_IF;


IF in_pressure < (set_pressure - histeresys) THEN
	work_time := TIME() - start_time;
	IF work_time >= delay_on THEN
		IF i = index_pivot AND index_pivot < len_active_pumps THEN
			i := i + 1;
		END_IF;
		cascade_pumps[index_active_pumps[i]].cascade_pump := TRUE;
		i := i + 1;
		start_time := t#0s;
	END_IF;
ELSIF in_pressure > (set_pressure + histeresys) THEN
	work_time := TIME() - start_time;
	IF work_time >= delay_off THEN
		IF i = index_pivot AND index_pivot > 1 THEN
			i := i - 1;
		END_IF;
		cascade_pumps[index_active_pumps[i]].cascade_pump := FALSE;
		i := i - 1;
		start_time := t#0s;
	END_IF;
END_IF;

